(* PLC project marvel_thermoVac, Institute of Astronomy Onto 0.0.1 *)
(* stored: creationDateTime 2025-01-01T00:00:00.0, modificationDateTime 2025-01-01T00:00:00.0 *)

{attribute 'qualified_only'}
TYPE TempControlStates : (idle := 0, warming_up := 1, unstable := 2, controlled := 3);
END_TYPE

{attribute 'qualified_only'}
TYPE TempControlStatus : (unknown := 0, invalid_model := 1, idle := 2, warming_up := 3, unstable := 4, controlled := 5) BYTE;
END_TYPE

TYPE InnerRoomControlParts : STRUCT
  {attribute 'TcHmiSymbol.Show'}
  tpT1 : TempMeasurement;  (* 1st temp sensor *)
  {attribute 'TcHmiSymbol.Show'}
  tpT2 : TempMeasurement;  (* 2nd temp sensor *)
  {attribute 'TcHmiSymbol.Show'}
  tpT3 : TempMeasurement;  (* 3rd temp sensor *)
  {attribute 'TcHmiSymbol.Show'}
  tpT4 : TempMeasurement;  (* 4th temp sensor *)
END_STRUCT;
END_TYPE

TYPE VesselControlParts : STRUCT
  {attribute 'TcHmiSymbol.Show'}
  tpLegNE : TempMeasurement;  (* Leg NE *)
  {attribute 'TcHmiSymbol.Show'}
  tpLegNW : TempMeasurement;  (* Leg NW *)
  {attribute 'TcHmiSymbol.Show'}
  tpLegSE : TempMeasurement;  (* Leg SE *)
  {attribute 'TcHmiSymbol.Show'}
  tpLegSW : TempMeasurement;  (* Leg SW *)
  {attribute 'TcHmiSymbol.Show'}
  tpLegTopNE : TempMeasurement;  (* Leg Top NE *)
  {attribute 'TcHmiSymbol.Show'}
  tpLegTopNW : TempMeasurement;  (* Leg Top NW *)
  {attribute 'TcHmiSymbol.Show'}
  tpLegTopSE : TempMeasurement;  (* Leg Top SE *)
  {attribute 'TcHmiSymbol.Show'}
  tpLegTopSW : TempMeasurement;  (* Leg Top SW *)
  {attribute 'TcHmiSymbol.Show'}
  tpVesBotNE : TempMeasurement;  (* Vessel Bottom NE *)
  {attribute 'TcHmiSymbol.Show'}
  tpVesBotNW : TempMeasurement;  (* Vessel Bottom NW *)
  {attribute 'TcHmiSymbol.Show'}
  tpVesBotSE : TempMeasurement;  (* Vessel Bottom SE *)
  {attribute 'TcHmiSymbol.Show'}
  tpVesBotSW : TempMeasurement;  (* Vessel Bottom SW *)
  {attribute 'TcHmiSymbol.Show'}
  tpCentre : TempMeasurement;  (* Centre *)
  {attribute 'TcHmiSymbol.Show'}
  tpCentreTH10K : TempMeasurement;  (* Centre TH10K *)
  {attribute 'TcHmiSymbol.Show'}
  tpVesSideN : TempMeasurement;  (* Vessel Side N *)
  {attribute 'TcHmiSymbol.Show'}
  tpVesSideS : TempMeasurement;  (* Vessel Side S *)
  {attribute 'TcHmiSymbol.Show'}
  tpVesSideE : TempMeasurement;  (* Vessel Side E *)
  {attribute 'TcHmiSymbol.Show'}
  tpVesSideW : TempMeasurement;  (* Vessel Side W *)
  {attribute 'TcHmiSymbol.Show'}
  tpVesLidN : TempMeasurement;  (* Vessel Lid N *)
  {attribute 'TcHmiSymbol.Show'}
  tpVesLidS : TempMeasurement;  (* Vessel Lid S *)
  {attribute 'TcHmiSymbol.Show'}
  htLegNE : HeaterControl;  (* Heater control for Leg NE *)
  {attribute 'TcHmiSymbol.Show'}
  htLegNW : HeaterControl;  (* Heater control for Leg NW *)
  {attribute 'TcHmiSymbol.Show'}
  htLegSE : HeaterControl;  (* Heater control for Leg SE *)
  {attribute 'TcHmiSymbol.Show'}
  htLegSW : HeaterControl;  (* Heater control for Leg SW *)
  {attribute 'TcHmiSymbol.Show'}
  htLegTopNE : HeaterControl;  (* Heater control for Leg Top NE *)
  {attribute 'TcHmiSymbol.Show'}
  htLegTopNW : HeaterControl;  (* Heater control for Leg Top NW *)
  {attribute 'TcHmiSymbol.Show'}
  htLegTopSE : HeaterControl;  (* Heater control for Leg Top SE *)
  {attribute 'TcHmiSymbol.Show'}
  htLegTopSW : HeaterControl;  (* Heater control for Leg Top SW *)
  {attribute 'TcHmiSymbol.Show'}
  htVesBotNE : HeaterControl;  (* Heater control for Vessel Bottom NE *)
  {attribute 'TcHmiSymbol.Show'}
  htVesBotNW : HeaterControl;  (* Heater control for Vessel Bottom NW *)
  {attribute 'TcHmiSymbol.Show'}
  htVesBotSE : HeaterControl;  (* Heater control for Vessel Bottom SE *)
  {attribute 'TcHmiSymbol.Show'}
  htVesBotSW : HeaterControl;  (* Heater control for Vessel Bottom SW *)
  {attribute 'TcHmiSymbol.Show'}
  htVesSideN : HeaterControl;  (* Heater control for Vessel Side NE *)
  {attribute 'TcHmiSymbol.Show'}
  htVesSideS : HeaterControl;  (* Heater control for Vessel Side NW *)
  {attribute 'TcHmiSymbol.Show'}
  htVesSideE : HeaterControl;  (* Heater control for Vessel Side SE *)
  {attribute 'TcHmiSymbol.Show'}
  htVesSideW : HeaterControl;  (* Heater control for Vessel Side SW *)
  {attribute 'TcHmiSymbol.Show'}
  htVesLidN : HeaterControl;  (* Heater control for Vessel Lid N *)
  {attribute 'TcHmiSymbol.Show'}
  htVesLidS : HeaterControl;  (* Heater control for Vessel Lid S *)
END_STRUCT;
END_TYPE

TYPE CryoControlParts : STRUCT
  {attribute 'TcHmiSymbol.Show'}
  tpCryoRear : TempMeasurement;  (* temp cryo rear / outside *)
  {attribute 'TcHmiSymbol.Show'}
  htCryoRear : HeaterControl;  (* heater cryo rear / outside *)
END_STRUCT;
END_TYPE

TYPE ThermoControlParts : STRUCT
  {attribute 'TcHmiSymbol.Show'}
  vessel : VesselControl;  (* State machine for the vessel temperature control *)
  {attribute 'TcHmiSymbol.Show'}
  innerRoom : InnerRoomControl;  (* State machine for the inner room temperature control *)
  {attribute 'TcHmiSymbol.Show'}
  configManager : ConfigManager;  (* The config manager (to load/save/activate configuration data) *)
END_STRUCT;
END_TYPE

TYPE HeaterControlProcesses : STRUCT
  {attribute 'TcHmiSymbol.Show'}
  initialize : Process;  (* Initialize the heater *)
  {attribute 'TcHmiSymbol.Show'}
  reset : Process;  (* Reset the heater *)
END_STRUCT;
END_TYPE

TYPE OuterRoomControlProcesses : STRUCT
  {attribute 'TcHmiSymbol.Show'}
  initialize : Process;  (* Start initializing *)
  {attribute 'TcHmiSymbol.Show'}
  start : Process;  (* Start warming up *)
  {attribute 'TcHmiSymbol.Show'}
  stop : Process;  (* Stop heating *)
  {attribute 'TcHmiSymbol.Show'}
  reset : Process;  (* Reset complete *)
  {attribute 'TcHmiSymbol.Show'}
  lock : Process;  (* Lock the outer room control (e.g. when the outer room is opened) *)
  {attribute 'TcHmiSymbol.Show'}
  unlock : Process;  (* Unlock the outer room control (e.g. when the outer room is closed) *)
END_STRUCT;
END_TYPE

TYPE InnerRoomControlProcesses : STRUCT
  {attribute 'TcHmiSymbol.Show'}
  initialize : Process;  (* Start initializing *)
  {attribute 'TcHmiSymbol.Show'}
  start : Process;  (* Start warming up *)
  {attribute 'TcHmiSymbol.Show'}
  stop : Process;  (* Stop heating *)
  {attribute 'TcHmiSymbol.Show'}
  reset : Process;  (* Reset complete *)
  {attribute 'TcHmiSymbol.Show'}
  lock : Process;  (* Lock the vessel control (e.g. when the vessel is opened) *)
  {attribute 'TcHmiSymbol.Show'}
  unlock : Process;  (* Unlock the vessel control (e.g. when the vessel is closed) *)
END_STRUCT;
END_TYPE

TYPE VesselControlProcesses : STRUCT
  {attribute 'TcHmiSymbol.Show'}
  initialize : Process;  (* Start initializing *)
  {attribute 'TcHmiSymbol.Show'}
  start : Process;  (* Start warming up *)
  {attribute 'TcHmiSymbol.Show'}
  stop : Process;  (* Stop heating *)
  {attribute 'TcHmiSymbol.Show'}
  reset : Process;  (* Reset complete *)
  {attribute 'TcHmiSymbol.Show'}
  lock : Process;  (* Lock the vessel control (e.g. when the vessel is opened) *)
  {attribute 'TcHmiSymbol.Show'}
  unlock : Process;  (* Unlock the vessel control (e.g. when the vessel is closed) *)
END_STRUCT;
END_TYPE

TYPE ShieldControlProcesses : STRUCT
  {attribute 'TcHmiSymbol.Show'}
  initialize : Process;  (* Start initializing *)
  {attribute 'TcHmiSymbol.Show'}
  start : Process;  (* Start warming up *)
  {attribute 'TcHmiSymbol.Show'}
  stop : Process;  (* Stop heating *)
  {attribute 'TcHmiSymbol.Show'}
  reset : Process;  (* Reset complete *)
  {attribute 'TcHmiSymbol.Show'}
  lock : Process;  (* Lock the shield control (e.g. when the shield is opened) *)
  {attribute 'TcHmiSymbol.Show'}
  unlock : Process;  (* Unlock the shield control (e.g. when the shield is closed) *)
END_STRUCT;
END_TYPE

TYPE BenchControlProcesses : STRUCT
  {attribute 'TcHmiSymbol.Show'}
  initialize : Process;  (* Start initializing *)
  {attribute 'TcHmiSymbol.Show'}
  start : Process;  (* Start warming up *)
  {attribute 'TcHmiSymbol.Show'}
  stop : Process;  (* Stop heating *)
  {attribute 'TcHmiSymbol.Show'}
  reset : Process;  (* Reset complete *)
  {attribute 'TcHmiSymbol.Show'}
  lock : Process;  (* Lock the bench control (e.g. when the bench is opened) *)
  {attribute 'TcHmiSymbol.Show'}
  unlock : Process;  (* Unlock the bench control (e.g. when the bench is closed) *)
END_STRUCT;
END_TYPE

TYPE CryoControlProcesses : STRUCT
  {attribute 'TcHmiSymbol.Show'}
  initialize : Process;  (* Start initializing *)
  {attribute 'TcHmiSymbol.Show'}
  start : Process;  (* Start warming up *)
  {attribute 'TcHmiSymbol.Show'}
  stop : Process;  (* Stop heating *)
  {attribute 'TcHmiSymbol.Show'}
  reset : Process;  (* Reset complete *)
  {attribute 'TcHmiSymbol.Show'}
  lock : Process;  (* Lock the bench control (e.g. when the bench is opened) *)
  {attribute 'TcHmiSymbol.Show'}
  unlock : Process;  (* Unlock the bench control (e.g. when the bench is closed) *)
END_STRUCT;
END_TYPE

TYPE ThermoControlProcesses : STRUCT
  {attribute 'TcHmiSymbol.Show'}
  initialize : Process;  (* Start initializing *)
  {attribute 'TcHmiSymbol.Show'}
  start : Process;  (* Start warming up *)
  {attribute 'TcHmiSymbol.Show'}
  stop : Process;  (* Stop heating *)
  {attribute 'TcHmiSymbol.Show'}
  reset : Process;  (* Reset complete *)
  {attribute 'TcHmiSymbol.Show'}
  lock : Process;  (* Lock the vessel control (e.g. when the vessel is opened) *)
  {attribute 'TcHmiSymbol.Show'}
  unlock : Process;  (* Unlock the vessel control (e.g. when the vessel is closed) *)
END_STRUCT;
END_TYPE

TYPE TempMeasurementStatuses : STRUCT
  {attribute 'OPC.UA.DA' := '1'}
  {attribute 'OPC.UA.DA.Access' := '1'}
  {attribute 'TcHmiSymbol.Show'}
  enabled : EnabledStatus;  (* Is the measurement enabled? *)
  {attribute 'OPC.UA.DA' := '1'}
  {attribute 'OPC.UA.DA.Access' := '1'}
  {attribute 'TcHmiSymbol.Show'}
  health : HealthStatus;  (* Is the measurement OK? *)
  {attribute 'OPC.UA.DA' := '1'}
  {attribute 'OPC.UA.DA.Access' := '1'}
  {attribute 'TcHmiSymbol.Show'}
  alarm : HiHiLoLoAlarmStatus;  (* Alarm status *)
END_STRUCT;
END_TYPE

TYPE HeaterControlStatuses : STRUCT
  {attribute 'OPC.UA.DA' := '1'}
  {attribute 'OPC.UA.DA.Access' := '1'}
  {attribute 'TcHmiSymbol.Show'}
  init : InitializationStatus;
  {attribute 'OPC.UA.DA' := '1'}
  {attribute 'OPC.UA.DA.Access' := '1'}
  {attribute 'TcHmiSymbol.Show'}
  enabled : EnabledStatus;  (* Is the heater enabled? *)
  {attribute 'OPC.UA.DA' := '1'}
  {attribute 'OPC.UA.DA.Access' := '1'}
  {attribute 'TcHmiSymbol.Show'}
  health : HealthStatus;  (* Is the heater healthy? *)
END_STRUCT;
END_TYPE

TYPE OuterRoomControlStatuses : STRUCT
  {attribute 'OPC.UA.DA' := '1'}
  {attribute 'OPC.UA.DA.Access' := '1'}
  {attribute 'TcHmiSymbol.Show'}
  init : InitializationStatus;
  {attribute 'OPC.UA.DA' := '1'}
  {attribute 'OPC.UA.DA.Access' := '1'}
  {attribute 'TcHmiSymbol.Show'}
  health : HealthStatus;  (* Is the outer room healthy? *)
  {attribute 'OPC.UA.DA' := '1'}
  {attribute 'OPC.UA.DA.Access' := '1'}
  {attribute 'TcHmiSymbol.Show'}
  control : TempControlStatus;  (* Actual state of the outer room *)
  {attribute 'OPC.UA.DA' := '1'}
  {attribute 'OPC.UA.DA.Access' := '1'}
  {attribute 'TcHmiSymbol.Show'}
  busy : BusyStatus;  (* Is the outer room busy with a procedure? *)
END_STRUCT;
END_TYPE

TYPE InnerRoomControlStatuses : STRUCT
  {attribute 'OPC.UA.DA' := '1'}
  {attribute 'OPC.UA.DA.Access' := '1'}
  {attribute 'TcHmiSymbol.Show'}
  init : InitializationStatus;
  {attribute 'OPC.UA.DA' := '1'}
  {attribute 'OPC.UA.DA.Access' := '1'}
  {attribute 'TcHmiSymbol.Show'}
  health : HealthStatus;  (* Is the vessel healthy? *)
  {attribute 'OPC.UA.DA' := '1'}
  {attribute 'OPC.UA.DA.Access' := '1'}
  {attribute 'TcHmiSymbol.Show'}
  control : TempControlStatus;  (* Actual state of the vessel *)
  {attribute 'OPC.UA.DA' := '1'}
  {attribute 'OPC.UA.DA.Access' := '1'}
  {attribute 'TcHmiSymbol.Show'}
  busy : BusyStatus;  (* Is the vessel busy with a procedure? *)
END_STRUCT;
END_TYPE

TYPE VesselControlStatuses : STRUCT
  {attribute 'OPC.UA.DA' := '1'}
  {attribute 'OPC.UA.DA.Access' := '1'}
  {attribute 'TcHmiSymbol.Show'}
  init : InitializationStatus;
  {attribute 'OPC.UA.DA' := '1'}
  {attribute 'OPC.UA.DA.Access' := '1'}
  {attribute 'TcHmiSymbol.Show'}
  health : HealthStatus;  (* Is the vessel healthy? *)
  {attribute 'OPC.UA.DA' := '1'}
  {attribute 'OPC.UA.DA.Access' := '1'}
  {attribute 'TcHmiSymbol.Show'}
  control : TempControlStatus;  (* Actual state of the vessel *)
  {attribute 'OPC.UA.DA' := '1'}
  {attribute 'OPC.UA.DA.Access' := '1'}
  {attribute 'TcHmiSymbol.Show'}
  busy : BusyStatus;  (* Is the vessel busy with a procedure? *)
END_STRUCT;
END_TYPE

TYPE ShieldControlStatuses : STRUCT
  {attribute 'OPC.UA.DA' := '1'}
  {attribute 'OPC.UA.DA.Access' := '1'}
  {attribute 'TcHmiSymbol.Show'}
  init : InitializationStatus;
  {attribute 'OPC.UA.DA' := '1'}
  {attribute 'OPC.UA.DA.Access' := '1'}
  {attribute 'TcHmiSymbol.Show'}
  health : HealthStatus;  (* Is the shield healthy? *)
  {attribute 'OPC.UA.DA' := '1'}
  {attribute 'OPC.UA.DA.Access' := '1'}
  {attribute 'TcHmiSymbol.Show'}
  control : TempControlStatus;  (* Actual state of the shield *)
  {attribute 'OPC.UA.DA' := '1'}
  {attribute 'OPC.UA.DA.Access' := '1'}
  {attribute 'TcHmiSymbol.Show'}
  busy : BusyStatus;  (* Is the shield busy with a procedure? *)
END_STRUCT;
END_TYPE

TYPE BenchControlStatuses : STRUCT
  {attribute 'OPC.UA.DA' := '1'}
  {attribute 'OPC.UA.DA.Access' := '1'}
  {attribute 'TcHmiSymbol.Show'}
  init : InitializationStatus;
  {attribute 'OPC.UA.DA' := '1'}
  {attribute 'OPC.UA.DA.Access' := '1'}
  {attribute 'TcHmiSymbol.Show'}
  health : HealthStatus;  (* Is the bench healthy? *)
  {attribute 'OPC.UA.DA' := '1'}
  {attribute 'OPC.UA.DA.Access' := '1'}
  {attribute 'TcHmiSymbol.Show'}
  control : TempControlStatus;  (* Actual state of the bench *)
  {attribute 'OPC.UA.DA' := '1'}
  {attribute 'OPC.UA.DA.Access' := '1'}
  {attribute 'TcHmiSymbol.Show'}
  busy : BusyStatus;  (* Is the bench busy with a procedure? *)
END_STRUCT;
END_TYPE

TYPE CryoControlStatuses : STRUCT
  {attribute 'OPC.UA.DA' := '1'}
  {attribute 'OPC.UA.DA.Access' := '1'}
  {attribute 'TcHmiSymbol.Show'}
  init : InitializationStatus;
  {attribute 'OPC.UA.DA' := '1'}
  {attribute 'OPC.UA.DA.Access' := '1'}
  {attribute 'TcHmiSymbol.Show'}
  health : HealthStatus;  (* Is the bench healthy? *)
  {attribute 'OPC.UA.DA' := '1'}
  {attribute 'OPC.UA.DA.Access' := '1'}
  {attribute 'TcHmiSymbol.Show'}
  control : TempControlStatus;  (* Actual state of the bench *)
  {attribute 'OPC.UA.DA' := '1'}
  {attribute 'OPC.UA.DA.Access' := '1'}
  {attribute 'TcHmiSymbol.Show'}
  busy : BusyStatus;  (* Is the bench busy with a procedure? *)
END_STRUCT;
END_TYPE

TYPE ThermoControlStatuses : STRUCT
  {attribute 'OPC.UA.DA' := '1'}
  {attribute 'OPC.UA.DA.Access' := '1'}
  {attribute 'TcHmiSymbol.Show'}
  init : InitializationStatus;
  {attribute 'OPC.UA.DA' := '1'}
  {attribute 'OPC.UA.DA.Access' := '1'}
  {attribute 'TcHmiSymbol.Show'}
  health : HealthStatus;  (* Is the vessel healthy? *)
  {attribute 'OPC.UA.DA' := '1'}
  {attribute 'OPC.UA.DA.Access' := '1'}
  {attribute 'TcHmiSymbol.Show'}
  control : TempControlStatus;  (* Actual state of the vessel *)
  {attribute 'OPC.UA.DA' := '1'}
  {attribute 'OPC.UA.DA.Access' := '1'}
  {attribute 'TcHmiSymbol.Show'}
  busy : BusyStatus;  (* Is the vessel busy with a procedure? *)
END_STRUCT;
END_TYPE

TYPE HeaterConfig : STRUCT
  {attribute 'TcHmiSymbol.Show'}
  enabled : BOOL := TRUE;  (* True if the heater is enabled *)
  {attribute 'TcHmiSymbol.Show'}
  maxPower : LREAL := 100.0;  (* Maximum power of the heater *)
  {attribute 'TcHmiSymbol.Show'}
  Kp : LREAL;  (* proportional gain *)
  {attribute 'TcHmiSymbol.Show'}
  Tn : LREAL;  (* integral gain (in seconds) *)
  {attribute 'TcHmiSymbol.Show'}
  Tv : LREAL;  (* derivative gain D-T1 (in seconds) *)
  {attribute 'TcHmiSymbol.Show'}
  Td : LREAL;  (* derivative damping time D-T1 (in seconds) *)
END_STRUCT;
END_TYPE

TYPE MeasurementConfig2 : STRUCT
  {attribute 'TcHmiSymbol.Show'}
  enabled : BOOL := TRUE;  (* Is the quantity being measured? (Can be false e.g. if the sensor is deliberately not connected (yet).) *)
  {attribute 'TcHmiSymbol.Show'}
  gain : LREAL := 1.0;  (* Gain to be applied to the measured value (default: 1 = no gain) *)
  {attribute 'TcHmiSymbol.Show'}
  offset : LREAL;  (* Offset to be added to the measured value (default: 0 = no offset) *)
END_STRUCT;
END_TYPE

TYPE SimulationConfig : STRUCT
  {attribute 'TcHmiSymbol.Show'}
  ambient : LREAL;  (* starting temp of sensors *)
  {attribute 'TcHmiSymbol.Show'}
  heating : LREAL;  (* heating gain/factor (0-1) *)
  {attribute 'TcHmiSymbol.Show'}
  cooling : LREAL;  (* cooling factor (0-1) *)
  {attribute 'TcHmiSymbol.Show'}
  noise : LREAL;  (* factor (0-1) multiplied with random number (0-1) to create noise in the simulated temperature *)
END_STRUCT;
END_TYPE

TYPE SharedHeaterConfig : STRUCT
  {attribute 'TcHmiSymbol.Show'}
  hihiDeviation : LREAL;  (* max dev from setpoint *)
  {attribute 'TcHmiSymbol.Show'}
  hiDeviation : LREAL;  (* warning dev from setpoint *)
  {attribute 'TcHmiSymbol.Show'}
  maxPower : LREAL := 100.0;  (* Maximum total power of all heaters in percentage *)
  {attribute 'TcHmiSymbol.Show'}
  simulation : SimulationConfig;
END_STRUCT;
END_TYPE

TYPE OuterRoomSharedConfig : STRUCT
  {attribute 'TcHmiSymbol.Show'}
  sensors : HiHiLoLoAlarmConfig;  (* Alarm config for the temperature sensors in the outer room *)
END_STRUCT;
END_TYPE

TYPE InnerRoomSharedConfig : STRUCT
  {attribute 'TcHmiSymbol.Show'}
  sensors : HiHiLoLoAlarmConfig;  (* Alarm config for the temperature sensors in the inner room *)
END_STRUCT;
END_TYPE

TYPE VesselSharedConfig : STRUCT
  {attribute 'TcHmiSymbol.Show'}
  sensors : HiHiLoLoAlarmConfig;  (* Alarm config for the temperature sensors in the vessel *)
  {attribute 'TcHmiSymbol.Show'}
  heaters : SharedHeaterConfig;  (* Shared config for the heaters in the vessel *)
END_STRUCT;
END_TYPE

TYPE ShieldSharedConfig : STRUCT
  {attribute 'TcHmiSymbol.Show'}
  sensors : HiHiLoLoAlarmConfig;  (* Alarm config for the temperature sensors in the shield *)
END_STRUCT;
END_TYPE

TYPE BenchSharedConfig : STRUCT
  {attribute 'TcHmiSymbol.Show'}
  sensors : HiHiLoLoAlarmConfig;  (* Alarm config for the temperature sensors in the bench *)
END_STRUCT;
END_TYPE

TYPE CryoSharedConfig : STRUCT
  {attribute 'TcHmiSymbol.Show'}
  sensors : HiHiLoLoAlarmConfig;  (* Alarm config for the temperature sensors in the cryo *)
  {attribute 'TcHmiSymbol.Show'}
  heaters : SharedHeaterConfig;  (* Shared config for the heaters in the cryo *)
END_STRUCT;
END_TYPE

TYPE ThermoSharedConfig : STRUCT
  {attribute 'TcHmiSymbol.Show'}
  bool : BOOL;  (* place holder, shared config currently not used *)
END_STRUCT;
END_TYPE

TYPE OuterRoomConfig : STRUCT
  {attribute 'TcHmiSymbol.Show'}
  shared : OuterRoomSharedConfig;  (* Shared config for the outer room *)
END_STRUCT;
END_TYPE

TYPE InnerRoomConfig : STRUCT
  {attribute 'TcHmiSymbol.Show'}
  tpT1 : MeasurementConfig2;  (* Config for temp sensor T1 *)
  {attribute 'TcHmiSymbol.Show'}
  tpT2 : MeasurementConfig2;  (* Config for temp sensor T2 *)
  {attribute 'TcHmiSymbol.Show'}
  tpT3 : MeasurementConfig2;  (* Config for temp sensor T3 *)
  {attribute 'TcHmiSymbol.Show'}
  tpT4 : MeasurementConfig2;  (* Config for temp sensor T4 *)
  {attribute 'TcHmiSymbol.Show'}
  shared : InnerRoomSharedConfig;  (* Shared config for the inner room *)
END_STRUCT;
END_TYPE

TYPE VesselConfig : STRUCT
  {attribute 'TcHmiSymbol.Show'}
  isSimulated : BOOL;  (* True if the vessel temperature control is in simulation mode *)
  {attribute 'TcHmiSymbol.Show'}
  setPointTarget : LREAL;  (* set point temperature in kelvin *)
  {attribute 'TcHmiSymbol.Show'}
  rampVPos : LREAL;  (* velocity of temperature change in K/s while ramping up *)
  {attribute 'TcHmiSymbol.Show'}
  rampVNeg : LREAL;  (* velocity of temperature change in K/s while ramping down *)
  {attribute 'TcHmiSymbol.Show'}
  rampStart : LREAL;  (* temperature in kelvin at which the ramp starts (e.g. to avoid overshoot) *)
  {attribute 'TcHmiSymbol.Show'}
  hihiDeviation : LREAL;  (* max dev from setpoint for the vessel *)
  {attribute 'TcHmiSymbol.Show'}
  hiDeviation : LREAL;  (* warning dev from setpoint for the vessel *)
  {attribute 'TcHmiSymbol.Show'}
  shared : VesselSharedConfig;  (* Shared config for the vessel *)
  {attribute 'TcHmiSymbol.Show'}
  tpLegNE : MeasurementConfig2;  (* Config for Leg NE *)
  {attribute 'TcHmiSymbol.Show'}
  tpLegNW : MeasurementConfig2;  (* Config for Leg NW *)
  {attribute 'TcHmiSymbol.Show'}
  tpLegSE : MeasurementConfig2;  (* Config for Leg SE *)
  {attribute 'TcHmiSymbol.Show'}
  tpLegSW : MeasurementConfig2;  (* Config for Leg SW *)
  {attribute 'TcHmiSymbol.Show'}
  tpLegTopNE : MeasurementConfig2;  (* Config for Leg Top NE *)
  {attribute 'TcHmiSymbol.Show'}
  tpLegTopNW : MeasurementConfig2;  (* Config for Leg Top NW *)
  {attribute 'TcHmiSymbol.Show'}
  tpLegTopSE : MeasurementConfig2;  (* Config for Leg Top SE *)
  {attribute 'TcHmiSymbol.Show'}
  tpLegTopSW : MeasurementConfig2;  (* Config for Leg Top SW *)
  {attribute 'TcHmiSymbol.Show'}
  tpVesBotNE : MeasurementConfig2;  (* Config for Vessel Bottom NE *)
  {attribute 'TcHmiSymbol.Show'}
  tpVesBotNW : MeasurementConfig2;  (* Config for Vessel Bottom NW *)
  {attribute 'TcHmiSymbol.Show'}
  tpVesBotSE : MeasurementConfig2;  (* Config for Vessel Bottom SE *)
  {attribute 'TcHmiSymbol.Show'}
  tpVesBotSW : MeasurementConfig2;  (* Config for Vessel Bottom SW *)
  {attribute 'TcHmiSymbol.Show'}
  tpCentre : MeasurementConfig2;  (* Config for Centre *)
  {attribute 'TcHmiSymbol.Show'}
  tpCentreTH10K : MeasurementConfig2;  (* Config for Centre TH10K *)
  {attribute 'TcHmiSymbol.Show'}
  tpVesSideN : MeasurementConfig2;  (* Config for Vessel Side N *)
  {attribute 'TcHmiSymbol.Show'}
  tpVesSideS : MeasurementConfig2;  (* Config for Vessel Side S *)
  {attribute 'TcHmiSymbol.Show'}
  tpVesSideE : MeasurementConfig2;  (* Config for Vessel Side E *)
  {attribute 'TcHmiSymbol.Show'}
  tpVesSideW : MeasurementConfig2;  (* Config for Vessel Side W *)
  {attribute 'TcHmiSymbol.Show'}
  tpVesLidN : MeasurementConfig2;  (* Config for Vessel Lid N *)
  {attribute 'TcHmiSymbol.Show'}
  tpVesLidS : MeasurementConfig2;  (* Config for Vessel Lid S *)
  {attribute 'TcHmiSymbol.Show'}
  htLegNE : HeaterConfig;  (* Config for heater Leg NE *)
  {attribute 'TcHmiSymbol.Show'}
  htLegNW : HeaterConfig;  (* Config for heater Leg NW *)
  {attribute 'TcHmiSymbol.Show'}
  htLegSE : HeaterConfig;  (* Config for heater Leg SE *)
  {attribute 'TcHmiSymbol.Show'}
  htLegSW : HeaterConfig;  (* Config for heater Leg SW *)
  {attribute 'TcHmiSymbol.Show'}
  htLegTopNE : HeaterConfig;  (* Config for heater Leg Top NE *)
  {attribute 'TcHmiSymbol.Show'}
  htLegTopNW : HeaterConfig;  (* Config for heater Leg Top NW *)
  {attribute 'TcHmiSymbol.Show'}
  htLegTopSE : HeaterConfig;  (* Config for heater Leg Top SE *)
  {attribute 'TcHmiSymbol.Show'}
  htLegTopSW : HeaterConfig;  (* Config for heater Leg Top SW *)
  {attribute 'TcHmiSymbol.Show'}
  htVesBotNE : HeaterConfig;  (* Config for heater Vessel Bottom NE *)
  {attribute 'TcHmiSymbol.Show'}
  htVesBotNW : HeaterConfig;  (* Config for heater Vessel Bottom NW *)
  {attribute 'TcHmiSymbol.Show'}
  htVesBotSE : HeaterConfig;  (* Config for heater Vessel Bottom SE *)
  {attribute 'TcHmiSymbol.Show'}
  htVesBotSW : HeaterConfig;  (* Config for heater Vessel Bottom SW *)
  {attribute 'TcHmiSymbol.Show'}
  htVesSideN : HeaterConfig;  (* Config for heater Vessel Side NE *)
  {attribute 'TcHmiSymbol.Show'}
  htVesSideS : HeaterConfig;  (* Config for heater Vessel Side NW *)
  {attribute 'TcHmiSymbol.Show'}
  htVesSideE : HeaterConfig;  (* Config for heater Vessel Side SE *)
  {attribute 'TcHmiSymbol.Show'}
  htVesSideW : HeaterConfig;  (* Config for heater Vessel Side SW *)
  {attribute 'TcHmiSymbol.Show'}
  htVesLidN : HeaterConfig;  (* Config for heater Vessel Lid N *)
  {attribute 'TcHmiSymbol.Show'}
  htVesLidS : HeaterConfig;  (* Config for heater Vessel Lid S *)
END_STRUCT;
END_TYPE

TYPE ShieldConfig : STRUCT
  {attribute 'TcHmiSymbol.Show'}
  shared : ShieldSharedConfig;  (* Shared config for the shield *)
END_STRUCT;
END_TYPE

TYPE BenchConfig : STRUCT
  {attribute 'TcHmiSymbol.Show'}
  shared : BenchSharedConfig;  (* Shared config for the bench *)
END_STRUCT;
END_TYPE

TYPE CryoConfig : STRUCT
  {attribute 'TcHmiSymbol.Show'}
  shared : CryoSharedConfig;  (* Shared config for the cryo *)
  {attribute 'TcHmiSymbol.Show'}
  tpCryoRear : MeasurementConfig2;  (* config for sensor cryo rear (outside) *)
  {attribute 'TcHmiSymbol.Show'}
  htCryoRear : HeaterConfig;  (* config for heater cryo rear (outside) *)
END_STRUCT;
END_TYPE

TYPE ThermoConfig : STRUCT
  {attribute 'TcHmiSymbol.Show'}
  outerRoom : OuterRoomConfig;  (* Config for the outer room *)
  {attribute 'TcHmiSymbol.Show'}
  innerRoom : InnerRoomConfig;  (* Config for the inner room *)
  {attribute 'TcHmiSymbol.Show'}
  vessel : VesselConfig;  (* Config for the vessel *)
  {attribute 'TcHmiSymbol.Show'}
  shield : ShieldConfig;  (* Config for the shield *)
  {attribute 'TcHmiSymbol.Show'}
  bench : BenchConfig;  (* Config for the bench *)
  {attribute 'TcHmiSymbol.Show'}
  cryo : CryoConfig;  (* Config for the cryo *)
  {attribute 'TcHmiSymbol.Show'}
  shared : ThermoSharedConfig;  (* Shared config for the thermo system *)
END_STRUCT;
END_TYPE

TYPE M_SM_TempMeasurement : STRUCT
  {attribute 'OPC.UA.DA' := '1'}
  {attribute 'OPC.UA.DA.Access' := '1'}
  {attribute 'TcHmiSymbol.Show'}
  isSimulated : BOOL;
  {attribute 'OPC.UA.DA' := '1'}
  {attribute 'OPC.UA.DA.Access' := '1'}
  {attribute 'TcHmiSymbol.Show'}
  simulatedVal : LREAL;
  {attribute 'OPC.UA.DA' := '1'}
  {attribute 'OPC.UA.DA.Access' := '1'}
  {attribute 'TcHmiSymbol.Show'}
  actualStatus : STRING;
  {attribute 'OPC.UA.DA' := '1'}
  {attribute 'OPC.UA.DA.Access' := '1'}
  {attribute 'TcHmiSymbol.Show'}
  actual : LREAL;
  {attribute 'OPC.UA.DA' := '1'}
  {attribute 'OPC.UA.DA.Access' := '1'}
  {attribute 'TcHmiSymbol.Show'}
  average : LREAL;
  {attribute 'OPC.UA.DA' := '1'}
  {attribute 'OPC.UA.DA.Access' := '1'}
  {attribute 'TcHmiSymbol.Show'}
  error : BOOL;
  {attribute 'OPC.UA.DA' := '1'}
  {attribute 'TcHmiSymbol.Show'}
  stat : TempMeasurementStatuses;
END_STRUCT;
END_TYPE

TYPE M_SM_HeaterControl : STRUCT
  {attribute 'OPC.UA.DA' := '1'}
  {attribute 'OPC.UA.DA.Access' := '1'}
  {attribute 'TcHmiSymbol.Show'}
  setPoint : LREAL;
  {attribute 'OPC.UA.DA' := '1'}
  {attribute 'OPC.UA.DA.Access' := '1'}
  {attribute 'TcHmiSymbol.Show'}
  temp : LREAL;
  {attribute 'OPC.UA.DA' := '1'}
  {attribute 'OPC.UA.DA.Access' := '1'}
  {attribute 'TcHmiSymbol.Show'}
  isSimulated : BOOL;
  {attribute 'OPC.UA.DA' := '1'}
  {attribute 'OPC.UA.DA.Access' := '1'}
  {attribute 'TcHmiSymbol.Show'}
  actualStatus : STRING;
  {attribute 'OPC.UA.DA' := '1'}
  {attribute 'OPC.UA.DA.Access' := '1'}
  {attribute 'TcHmiSymbol.Show'}
  power : LREAL;
  {attribute 'OPC.UA.DA' := '1'}
  {attribute 'OPC.UA.DA.Access' := '1'}
  {attribute 'TcHmiSymbol.Show'}
  active : BOOL;
  {attribute 'OPC.UA.DA' := '1'}
  {attribute 'OPC.UA.DA.Access' := '1'}
  {attribute 'TcHmiSymbol.Show'}
  deviation : LREAL;
  {attribute 'OPC.UA.DA' := '1'}
  {attribute 'OPC.UA.DA.Access' := '1'}
  {attribute 'TcHmiSymbol.Show'}
  isControlled : BOOL;
  {attribute 'OPC.UA.DA' := '1'}
  {attribute 'OPC.UA.DA.Access' := '1'}
  {attribute 'TcHmiSymbol.Show'}
  simTemp : LREAL;
  {attribute 'OPC.UA.DA' := '1'}
  {attribute 'TcHmiSymbol.Show'}
  stat : HeaterControlStatuses;
  {attribute 'OPC.UA.DA' := '1'}
  {attribute 'TcHmiSymbol.Show'}
  proc : M_SM_HeaterControlProcesses;
END_STRUCT;
END_TYPE

TYPE M_SM_OuterRoomControl : STRUCT
  {attribute 'OPC.UA.DA' := '1'}
  {attribute 'OPC.UA.DA.Access' := '1'}
  {attribute 'TcHmiSymbol.Show'}
  actualStatus : STRING;
  {attribute 'OPC.UA.DA' := '1'}
  {attribute 'OPC.UA.DA.Access' := '1'}
  {attribute 'TcHmiSymbol.Show'}
  avgTemp : LREAL;
  {attribute 'OPC.UA.DA' := '1'}
  {attribute 'OPC.UA.DA.Access' := '1'}
  {attribute 'TcHmiSymbol.Show'}
  maxDeviation : LREAL;
  {attribute 'OPC.UA.DA' := '1'}
  {attribute 'OPC.UA.DA.Access' := '1'}
  {attribute 'TcHmiSymbol.Show'}
  avgDeviation : LREAL;
  {attribute 'OPC.UA.DA' := '1'}
  {attribute 'OPC.UA.DA.Access' := '1'}
  {attribute 'TcHmiSymbol.Show'}
  totalPower : LREAL;
  {attribute 'OPC.UA.DA' := '1'}
  {attribute 'OPC.UA.DA.Access' := '1'}
  {attribute 'TcHmiSymbol.Show'}
  avgPower : LREAL;
  {attribute 'OPC.UA.DA' := '1'}
  {attribute 'TcHmiSymbol.Show'}
  stat : OuterRoomControlStatuses;
  {attribute 'OPC.UA.DA' := '1'}
  {attribute 'TcHmiSymbol.Show'}
  proc : M_SM_OuterRoomControlProcesses;
END_STRUCT;
END_TYPE

TYPE M_SM_InnerRoomControl : STRUCT
  {attribute 'OPC.UA.DA' := '1'}
  {attribute 'OPC.UA.DA.Access' := '1'}
  {attribute 'TcHmiSymbol.Show'}
  actualStatus : STRING;
  {attribute 'OPC.UA.DA' := '1'}
  {attribute 'OPC.UA.DA.Access' := '1'}
  {attribute 'TcHmiSymbol.Show'}
  avgTemp : LREAL;
  {attribute 'OPC.UA.DA' := '1'}
  {attribute 'OPC.UA.DA.Access' := '1'}
  {attribute 'TcHmiSymbol.Show'}
  maxDeviation : LREAL;
  {attribute 'OPC.UA.DA' := '1'}
  {attribute 'OPC.UA.DA.Access' := '1'}
  {attribute 'TcHmiSymbol.Show'}
  avgDeviation : LREAL;
  {attribute 'OPC.UA.DA' := '1'}
  {attribute 'OPC.UA.DA.Access' := '1'}
  {attribute 'TcHmiSymbol.Show'}
  totalPower : LREAL;
  {attribute 'OPC.UA.DA' := '1'}
  {attribute 'OPC.UA.DA.Access' := '1'}
  {attribute 'TcHmiSymbol.Show'}
  avgPower : LREAL;
  {attribute 'OPC.UA.DA' := '1'}
  {attribute 'TcHmiSymbol.Show'}
  stat : InnerRoomControlStatuses;
  {attribute 'OPC.UA.DA' := '1'}
  {attribute 'TcHmiSymbol.Show'}
  parts : M_SM_InnerRoomControlParts;
  {attribute 'OPC.UA.DA' := '1'}
  {attribute 'TcHmiSymbol.Show'}
  proc : M_SM_InnerRoomControlProcesses;
END_STRUCT;
END_TYPE

TYPE M_SM_VesselControl : STRUCT
  {attribute 'OPC.UA.DA' := '1'}
  {attribute 'OPC.UA.DA.Access' := '1'}
  {attribute 'TcHmiSymbol.Show'}
  tStatBottomOk : BOOL;
  {attribute 'OPC.UA.DA' := '1'}
  {attribute 'OPC.UA.DA.Access' := '1'}
  {attribute 'TcHmiSymbol.Show'}
  tStatCryoRearOk : BOOL;
  {attribute 'OPC.UA.DA' := '1'}
  {attribute 'OPC.UA.DA.Access' := '1'}
  {attribute 'TcHmiSymbol.Show'}
  tStatLidOk : BOOL;
  {attribute 'OPC.UA.DA' := '1'}
  {attribute 'OPC.UA.DA.Access' := '1'}
  {attribute 'TcHmiSymbol.Show'}
  actualStatus : STRING;
  {attribute 'OPC.UA.DA' := '1'}
  {attribute 'OPC.UA.DA.Access' := '1'}
  {attribute 'TcHmiSymbol.Show'}
  avgTemp : LREAL;
  {attribute 'OPC.UA.DA' := '1'}
  {attribute 'OPC.UA.DA.Access' := '1'}
  {attribute 'TcHmiSymbol.Show'}
  maxDeviation : LREAL;
  {attribute 'OPC.UA.DA' := '1'}
  {attribute 'OPC.UA.DA.Access' := '1'}
  {attribute 'TcHmiSymbol.Show'}
  avgDeviation : LREAL;
  {attribute 'OPC.UA.DA' := '1'}
  {attribute 'OPC.UA.DA.Access' := '1'}
  {attribute 'TcHmiSymbol.Show'}
  totalPower : LREAL;
  {attribute 'OPC.UA.DA' := '1'}
  {attribute 'OPC.UA.DA.Access' := '1'}
  {attribute 'TcHmiSymbol.Show'}
  avgPower : LREAL;
  {attribute 'OPC.UA.DA' := '1'}
  {attribute 'OPC.UA.DA.Access' := '1'}
  {attribute 'TcHmiSymbol.Show'}
  tStatBottomPwr : BOOL;
  {attribute 'OPC.UA.DA' := '1'}
  {attribute 'OPC.UA.DA.Access' := '1'}
  {attribute 'TcHmiSymbol.Show'}
  tStatCryoRearPwr : BOOL;
  {attribute 'OPC.UA.DA' := '1'}
  {attribute 'OPC.UA.DA.Access' := '1'}
  {attribute 'TcHmiSymbol.Show'}
  tStatLidPwr : BOOL;
  {attribute 'OPC.UA.DA' := '1'}
  {attribute 'TcHmiSymbol.Show'}
  stat : VesselControlStatuses;
  {attribute 'OPC.UA.DA' := '1'}
  {attribute 'TcHmiSymbol.Show'}
  parts : M_SM_VesselControlParts;
  {attribute 'OPC.UA.DA' := '1'}
  {attribute 'TcHmiSymbol.Show'}
  proc : M_SM_VesselControlProcesses;
END_STRUCT;
END_TYPE

TYPE M_SM_ShieldControl : STRUCT
  {attribute 'OPC.UA.DA' := '1'}
  {attribute 'OPC.UA.DA.Access' := '1'}
  {attribute 'TcHmiSymbol.Show'}
  actualStatus : STRING;
  {attribute 'OPC.UA.DA' := '1'}
  {attribute 'OPC.UA.DA.Access' := '1'}
  {attribute 'TcHmiSymbol.Show'}
  avgTemp : LREAL;
  {attribute 'OPC.UA.DA' := '1'}
  {attribute 'OPC.UA.DA.Access' := '1'}
  {attribute 'TcHmiSymbol.Show'}
  maxDeviation : LREAL;
  {attribute 'OPC.UA.DA' := '1'}
  {attribute 'OPC.UA.DA.Access' := '1'}
  {attribute 'TcHmiSymbol.Show'}
  avgDeviation : LREAL;
  {attribute 'OPC.UA.DA' := '1'}
  {attribute 'OPC.UA.DA.Access' := '1'}
  {attribute 'TcHmiSymbol.Show'}
  totalPower : LREAL;
  {attribute 'OPC.UA.DA' := '1'}
  {attribute 'OPC.UA.DA.Access' := '1'}
  {attribute 'TcHmiSymbol.Show'}
  avgPower : LREAL;
  {attribute 'OPC.UA.DA' := '1'}
  {attribute 'TcHmiSymbol.Show'}
  stat : ShieldControlStatuses;
  {attribute 'OPC.UA.DA' := '1'}
  {attribute 'TcHmiSymbol.Show'}
  proc : M_SM_ShieldControlProcesses;
END_STRUCT;
END_TYPE

TYPE M_SM_BenchControl : STRUCT
  {attribute 'OPC.UA.DA' := '1'}
  {attribute 'OPC.UA.DA.Access' := '1'}
  {attribute 'TcHmiSymbol.Show'}
  actualStatus : STRING;
  {attribute 'OPC.UA.DA' := '1'}
  {attribute 'OPC.UA.DA.Access' := '1'}
  {attribute 'TcHmiSymbol.Show'}
  avgTemp : LREAL;
  {attribute 'OPC.UA.DA' := '1'}
  {attribute 'OPC.UA.DA.Access' := '1'}
  {attribute 'TcHmiSymbol.Show'}
  maxDeviation : LREAL;
  {attribute 'OPC.UA.DA' := '1'}
  {attribute 'OPC.UA.DA.Access' := '1'}
  {attribute 'TcHmiSymbol.Show'}
  avgDeviation : LREAL;
  {attribute 'OPC.UA.DA' := '1'}
  {attribute 'OPC.UA.DA.Access' := '1'}
  {attribute 'TcHmiSymbol.Show'}
  totalPower : LREAL;
  {attribute 'OPC.UA.DA' := '1'}
  {attribute 'OPC.UA.DA.Access' := '1'}
  {attribute 'TcHmiSymbol.Show'}
  avgPower : LREAL;
  {attribute 'OPC.UA.DA' := '1'}
  {attribute 'TcHmiSymbol.Show'}
  stat : BenchControlStatuses;
  {attribute 'OPC.UA.DA' := '1'}
  {attribute 'TcHmiSymbol.Show'}
  proc : M_SM_BenchControlProcesses;
END_STRUCT;
END_TYPE

TYPE M_SM_CryoControl : STRUCT
  {attribute 'OPC.UA.DA' := '1'}
  {attribute 'OPC.UA.DA.Access' := '1'}
  {attribute 'TcHmiSymbol.Show'}
  actualStatus : STRING;
  {attribute 'OPC.UA.DA' := '1'}
  {attribute 'OPC.UA.DA.Access' := '1'}
  {attribute 'TcHmiSymbol.Show'}
  avgTemp : LREAL;
  {attribute 'OPC.UA.DA' := '1'}
  {attribute 'OPC.UA.DA.Access' := '1'}
  {attribute 'TcHmiSymbol.Show'}
  maxDeviation : LREAL;
  {attribute 'OPC.UA.DA' := '1'}
  {attribute 'OPC.UA.DA.Access' := '1'}
  {attribute 'TcHmiSymbol.Show'}
  avgDeviation : LREAL;
  {attribute 'OPC.UA.DA' := '1'}
  {attribute 'OPC.UA.DA.Access' := '1'}
  {attribute 'TcHmiSymbol.Show'}
  totalPower : LREAL;
  {attribute 'OPC.UA.DA' := '1'}
  {attribute 'OPC.UA.DA.Access' := '1'}
  {attribute 'TcHmiSymbol.Show'}
  avgPower : LREAL;
  {attribute 'OPC.UA.DA' := '1'}
  {attribute 'TcHmiSymbol.Show'}
  stat : CryoControlStatuses;
  {attribute 'OPC.UA.DA' := '1'}
  {attribute 'TcHmiSymbol.Show'}
  parts : M_SM_CryoControlParts;
  {attribute 'OPC.UA.DA' := '1'}
  {attribute 'TcHmiSymbol.Show'}
  proc : M_SM_CryoControlProcesses;
END_STRUCT;
END_TYPE

TYPE M_SM_ThermoControl : STRUCT
  {attribute 'OPC.UA.DA' := '1'}
  {attribute 'OPC.UA.DA.Access' := '3'}
  {attribute 'TcHmiSymbol.Show'}
  editableConfig : ThermoConfig;
  {attribute 'OPC.UA.DA' := '1'}
  {attribute 'OPC.UA.DA.Access' := '1'}
  {attribute 'TcHmiSymbol.Show'}
  actualStatus : STRING;
  {attribute 'OPC.UA.DA' := '1'}
  {attribute 'OPC.UA.DA.Access' := '1'}
  {attribute 'TcHmiSymbol.Show'}
  config : ThermoConfig;
  {attribute 'OPC.UA.DA' := '1'}
  {attribute 'OPC.UA.DA.Access' := '1'}
  {attribute 'TcHmiSymbol.Show'}
  setPointRamped : LREAL;
  {attribute 'OPC.UA.DA' := '1'}
  {attribute 'TcHmiSymbol.Show'}
  stat : ThermoControlStatuses;
  {attribute 'OPC.UA.DA' := '1'}
  {attribute 'TcHmiSymbol.Show'}
  parts : M_SM_ThermoControlParts;
  {attribute 'OPC.UA.DA' := '1'}
  {attribute 'TcHmiSymbol.Show'}
  proc : M_SM_ThermoControlProcesses;
END_STRUCT;
END_TYPE

TYPE M_SM_HeaterControlProcesses : STRUCT
  {attribute 'TcHmiSymbol.Show'}
  initialize : M_Process;
  {attribute 'TcHmiSymbol.Show'}
  reset : M_Process;
END_STRUCT;
END_TYPE

TYPE M_SM_OuterRoomControlProcesses : STRUCT
  {attribute 'TcHmiSymbol.Show'}
  initialize : M_Process;
  {attribute 'TcHmiSymbol.Show'}
  start : M_Process;
  {attribute 'TcHmiSymbol.Show'}
  stop : M_Process;
  {attribute 'TcHmiSymbol.Show'}
  reset : M_Process;
  {attribute 'TcHmiSymbol.Show'}
  lock : M_Process;
  {attribute 'TcHmiSymbol.Show'}
  unlock : M_Process;
END_STRUCT;
END_TYPE

TYPE M_SM_InnerRoomControlParts : STRUCT
  {attribute 'TcHmiSymbol.Show'}
  tpT1 : M_TempMeasurement;
  {attribute 'TcHmiSymbol.Show'}
  tpT2 : M_TempMeasurement;
  {attribute 'TcHmiSymbol.Show'}
  tpT3 : M_TempMeasurement;
  {attribute 'TcHmiSymbol.Show'}
  tpT4 : M_TempMeasurement;
END_STRUCT;
END_TYPE

TYPE M_SM_InnerRoomControlProcesses : STRUCT
  {attribute 'TcHmiSymbol.Show'}
  initialize : M_Process;
  {attribute 'TcHmiSymbol.Show'}
  start : M_Process;
  {attribute 'TcHmiSymbol.Show'}
  stop : M_Process;
  {attribute 'TcHmiSymbol.Show'}
  reset : M_Process;
  {attribute 'TcHmiSymbol.Show'}
  lock : M_Process;
  {attribute 'TcHmiSymbol.Show'}
  unlock : M_Process;
END_STRUCT;
END_TYPE

TYPE M_SM_VesselControlParts : STRUCT
  {attribute 'TcHmiSymbol.Show'}
  tpLegNE : M_TempMeasurement;
  {attribute 'TcHmiSymbol.Show'}
  tpLegNW : M_TempMeasurement;
  {attribute 'TcHmiSymbol.Show'}
  tpLegSE : M_TempMeasurement;
  {attribute 'TcHmiSymbol.Show'}
  tpLegSW : M_TempMeasurement;
  {attribute 'TcHmiSymbol.Show'}
  tpLegTopNE : M_TempMeasurement;
  {attribute 'TcHmiSymbol.Show'}
  tpLegTopNW : M_TempMeasurement;
  {attribute 'TcHmiSymbol.Show'}
  tpLegTopSE : M_TempMeasurement;
  {attribute 'TcHmiSymbol.Show'}
  tpLegTopSW : M_TempMeasurement;
  {attribute 'TcHmiSymbol.Show'}
  tpVesBotNE : M_TempMeasurement;
  {attribute 'TcHmiSymbol.Show'}
  tpVesBotNW : M_TempMeasurement;
  {attribute 'TcHmiSymbol.Show'}
  tpVesBotSE : M_TempMeasurement;
  {attribute 'TcHmiSymbol.Show'}
  tpVesBotSW : M_TempMeasurement;
  {attribute 'TcHmiSymbol.Show'}
  tpCentre : M_TempMeasurement;
  {attribute 'TcHmiSymbol.Show'}
  tpCentreTH10K : M_TempMeasurement;
  {attribute 'TcHmiSymbol.Show'}
  tpVesSideN : M_TempMeasurement;
  {attribute 'TcHmiSymbol.Show'}
  tpVesSideS : M_TempMeasurement;
  {attribute 'TcHmiSymbol.Show'}
  tpVesSideE : M_TempMeasurement;
  {attribute 'TcHmiSymbol.Show'}
  tpVesSideW : M_TempMeasurement;
  {attribute 'TcHmiSymbol.Show'}
  tpVesLidN : M_TempMeasurement;
  {attribute 'TcHmiSymbol.Show'}
  tpVesLidS : M_TempMeasurement;
  {attribute 'TcHmiSymbol.Show'}
  htLegNE : M_HeaterControl;
  {attribute 'TcHmiSymbol.Show'}
  htLegNW : M_HeaterControl;
  {attribute 'TcHmiSymbol.Show'}
  htLegSE : M_HeaterControl;
  {attribute 'TcHmiSymbol.Show'}
  htLegSW : M_HeaterControl;
  {attribute 'TcHmiSymbol.Show'}
  htLegTopNE : M_HeaterControl;
  {attribute 'TcHmiSymbol.Show'}
  htLegTopNW : M_HeaterControl;
  {attribute 'TcHmiSymbol.Show'}
  htLegTopSE : M_HeaterControl;
  {attribute 'TcHmiSymbol.Show'}
  htLegTopSW : M_HeaterControl;
  {attribute 'TcHmiSymbol.Show'}
  htVesBotNE : M_HeaterControl;
  {attribute 'TcHmiSymbol.Show'}
  htVesBotNW : M_HeaterControl;
  {attribute 'TcHmiSymbol.Show'}
  htVesBotSE : M_HeaterControl;
  {attribute 'TcHmiSymbol.Show'}
  htVesBotSW : M_HeaterControl;
  {attribute 'TcHmiSymbol.Show'}
  htVesSideN : M_HeaterControl;
  {attribute 'TcHmiSymbol.Show'}
  htVesSideS : M_HeaterControl;
  {attribute 'TcHmiSymbol.Show'}
  htVesSideE : M_HeaterControl;
  {attribute 'TcHmiSymbol.Show'}
  htVesSideW : M_HeaterControl;
  {attribute 'TcHmiSymbol.Show'}
  htVesLidN : M_HeaterControl;
  {attribute 'TcHmiSymbol.Show'}
  htVesLidS : M_HeaterControl;
END_STRUCT;
END_TYPE

TYPE M_SM_VesselControlProcesses : STRUCT
  {attribute 'TcHmiSymbol.Show'}
  initialize : M_Process;
  {attribute 'TcHmiSymbol.Show'}
  start : M_Process;
  {attribute 'TcHmiSymbol.Show'}
  stop : M_Process;
  {attribute 'TcHmiSymbol.Show'}
  reset : M_Process;
  {attribute 'TcHmiSymbol.Show'}
  lock : M_Process;
  {attribute 'TcHmiSymbol.Show'}
  unlock : M_Process;
END_STRUCT;
END_TYPE

TYPE M_SM_ShieldControlProcesses : STRUCT
  {attribute 'TcHmiSymbol.Show'}
  initialize : M_Process;
  {attribute 'TcHmiSymbol.Show'}
  start : M_Process;
  {attribute 'TcHmiSymbol.Show'}
  stop : M_Process;
  {attribute 'TcHmiSymbol.Show'}
  reset : M_Process;
  {attribute 'TcHmiSymbol.Show'}
  lock : M_Process;
  {attribute 'TcHmiSymbol.Show'}
  unlock : M_Process;
END_STRUCT;
END_TYPE

TYPE M_SM_BenchControlProcesses : STRUCT
  {attribute 'TcHmiSymbol.Show'}
  initialize : M_Process;
  {attribute 'TcHmiSymbol.Show'}
  start : M_Process;
  {attribute 'TcHmiSymbol.Show'}
  stop : M_Process;
  {attribute 'TcHmiSymbol.Show'}
  reset : M_Process;
  {attribute 'TcHmiSymbol.Show'}
  lock : M_Process;
  {attribute 'TcHmiSymbol.Show'}
  unlock : M_Process;
END_STRUCT;
END_TYPE

TYPE M_SM_CryoControlParts : STRUCT
  {attribute 'TcHmiSymbol.Show'}
  tpCryoRear : M_TempMeasurement;
  {attribute 'TcHmiSymbol.Show'}
  htCryoRear : M_HeaterControl;
END_STRUCT;
END_TYPE

TYPE M_SM_CryoControlProcesses : STRUCT
  {attribute 'TcHmiSymbol.Show'}
  initialize : M_Process;
  {attribute 'TcHmiSymbol.Show'}
  start : M_Process;
  {attribute 'TcHmiSymbol.Show'}
  stop : M_Process;
  {attribute 'TcHmiSymbol.Show'}
  reset : M_Process;
  {attribute 'TcHmiSymbol.Show'}
  lock : M_Process;
  {attribute 'TcHmiSymbol.Show'}
  unlock : M_Process;
END_STRUCT;
END_TYPE

TYPE M_SM_ThermoControlParts : STRUCT
  {attribute 'TcHmiSymbol.Show'}
  vessel : M_VesselControl;
  {attribute 'TcHmiSymbol.Show'}
  innerRoom : M_InnerRoomControl;
  {attribute 'TcHmiSymbol.Show'}
  configManager : M_ConfigManager;
END_STRUCT;
END_TYPE

TYPE M_SM_ThermoControlProcesses : STRUCT
  {attribute 'TcHmiSymbol.Show'}
  initialize : M_Process;
  {attribute 'TcHmiSymbol.Show'}
  start : M_Process;
  {attribute 'TcHmiSymbol.Show'}
  stop : M_Process;
  {attribute 'TcHmiSymbol.Show'}
  reset : M_Process;
  {attribute 'TcHmiSymbol.Show'}
  lock : M_Process;
  {attribute 'TcHmiSymbol.Show'}
  unlock : M_Process;
END_STRUCT;
END_TYPE

{attribute 'TcRpcEnable' := '1'}
FUNCTION F_TempControlStatus : TempControlStatus
  VAR_INPUT
    superState : BOOL := TRUE;  (* Super state (TRUE if the super state is active, or if there is no super state) *)
    isControlled : BOOL;  (* True if the vessel is in controlled state *)
    isActive : BOOL;  (* True if the vessel is active (not idle) *)
    isWarmingUp : BOOL;  (* True if the vessel is warming up *)
  END_VAR

              IF NOT(superState) THEN
    F_TempControlStatus := TempControlStatus.unknown;
ELSIF NOT(isActive) THEN
    F_TempControlStatus := TempControlStatus.idle;
ELSIF isActive AND isWarmingUp THEN
    F_TempControlStatus := TempControlStatus.warming_up;
ELSIF isActive AND ((NOT(isWarmingUp)) AND (NOT(isControlled))) THEN
    F_TempControlStatus := TempControlStatus.unstable;
ELSIF isActive AND ((NOT(isWarmingUp)) AND isControlled) THEN
    F_TempControlStatus := TempControlStatus.controlled;
ELSE
    F_TempControlStatus := TempControlStatus.invalid_model;
END_IF;

            
END_FUNCTION

FUNCTION_BLOCK SM_TempMeasurement
  VAR_INPUT
    {attribute 'OPC.UA.DA' := '1'}
    {attribute 'OPC.UA.DA.Access' := '1'}
    isSimulated : BOOL;
    {attribute 'OPC.UA.DA' := '1'}
    {attribute 'OPC.UA.DA.Access' := '1'}
    simulatedVal : LREAL;
    {attribute 'OPC.UA.DA' := '0'}
    rawValue AT %I* : REAL;  (* Measured raw value *)
    {attribute 'OPC.UA.DA' := '0'}
    conversionFactor : LREAL;  (* rawValue * conversionFactor = temperature.degrees.value *)
  END_VAR
  VAR_OUTPUT
    {attribute 'OPC.UA.DA' := '1'}
    {attribute 'OPC.UA.DA.Access' := '1'}
    actualStatus : STRING(50);  (* Current status description *)
    {attribute 'OPC.UA.DA' := '1'}
    {attribute 'OPC.UA.DA.Access' := '1'}
    actual : LREAL;  (* Actual value *)
    {attribute 'OPC.UA.DA' := '1'}
    {attribute 'OPC.UA.DA.Access' := '1'}
    average : LREAL;  (* Moving average value *)
    {attribute 'OPC.UA.DA' := '1'}
    {attribute 'OPC.UA.DA.Access' := '1'}
    error : BOOL;  (* true if there is an error *)
    {attribute 'OPC.UA.DA' := '1'}
    stat : TempMeasurementStatuses;  (* Statuses of the state machine *)
  END_VAR
  VAR_IN_OUT
    {attribute 'OPC.UA.DA' := '0'}
    config_ref : MeasurementConfig2;  (* Reference to the config (alarms in degrees celsius) *)
    {attribute 'OPC.UA.DA' := '0'}
    sharedConfig_ref : HiHiLoLoAlarmConfig;  (* Reference to the alarm config for the sensor *)
  END_VAR

            stat.enabled := F_EnabledStatus(
    superState := TRUE,
    isEnabled := config_ref.enabled);
stat.health := F_HealthStatus(
    superState := stat.enabled = EnabledStatus.enabled,
    isGood := NOT((stat.alarm = HiHiLoLoAlarmStatus.hiHi) OR ((stat.alarm = HiHiLoLoAlarmStatus.loLo) OR error)),
    hasWarning := (stat.alarm = HiHiLoLoAlarmStatus.hi) OR (stat.alarm = HiHiLoLoAlarmStatus.lo));

          

METHOD _copyFromModel_SM_TempMeasurement
  VAR_IN_OUT
    {attribute 'OPC.UA.DA' := '0'}
    model : M_SM_TempMeasurement;
  END_VAR
                  
                
END_METHOD

METHOD _copyToModel_SM_TempMeasurement
  VAR_IN_OUT
    {attribute 'OPC.UA.DA' := '0'}
    model : M_SM_TempMeasurement;
  END_VAR
                  model.isSimulated := THIS^.isSimulated;
model.simulatedVal := THIS^.simulatedVal;
model.actualStatus := THIS^.actualStatus;
model.actual := THIS^.actual;
model.average := THIS^.average;
model.error := THIS^.error;
model.stat := THIS^.stat;

                
END_METHOD
END_FUNCTION_BLOCK

FUNCTION_BLOCK SM_HeaterControl
  VAR_INPUT
    {attribute 'OPC.UA.DA' := '1'}
    {attribute 'OPC.UA.DA.Access' := '1'}
    setPoint : LREAL;  (* Current set point of the heater in kelvin *)
    {attribute 'OPC.UA.DA' := '1'}
    {attribute 'OPC.UA.DA.Access' := '1'}
    temp : LREAL;  (* Associated temperature of the heater in kelvin *)
    {attribute 'OPC.UA.DA' := '1'}
    {attribute 'OPC.UA.DA.Access' := '1'}
    isSimulated : BOOL;
  END_VAR
  VAR_OUTPUT
    {attribute 'OPC.UA.DA' := '1'}
    {attribute 'OPC.UA.DA.Access' := '1'}
    actualStatus : STRING(50);  (* Current status description *)
    {attribute 'OPC.UA.DA' := '1'}
    {attribute 'OPC.UA.DA.Access' := '1'}
    power : LREAL;  (* Current power of the heater in percentage *)
    {attribute 'OPC.UA.DA' := '1'}
    {attribute 'OPC.UA.DA.Access' := '1'}
    active : BOOL;  (* True if the heater is active *)
    {attribute 'OPC.UA.DA' := '1'}
    {attribute 'OPC.UA.DA.Access' := '1'}
    deviation : LREAL;  (* Current error between set point and associated temperature *)
    {attribute 'OPC.UA.DA' := '1'}
    {attribute 'OPC.UA.DA.Access' := '1'}
    isControlled : BOOL;  (* True if the heater is in controlled state *)
    {attribute 'OPC.UA.DA' := '1'}
    {attribute 'OPC.UA.DA.Access' := '1'}
    simTemp : LREAL;  (* Simulated temperature for testing the heater control *)
    {attribute 'OPC.UA.DA' := '1'}
    stat : HeaterControlStatuses;  (* Statuses of the state machine *)
    {attribute 'OPC.UA.DA' := '1'}
    proc : HeaterControlProcesses;  (* Processes of the state machine *)
  END_VAR
  VAR_IN_OUT
    {attribute 'OPC.UA.DA' := '0'}
    config_ref : HeaterConfig;  (* Reference to the heater config *)
    {attribute 'OPC.UA.DA' := '0'}
    sharedConfig_ref : SharedHeaterConfig;  (* Reference to the shared heater config *)
  END_VAR

            stat.enabled := F_EnabledStatus(
    superState := TRUE,
    isEnabled := config_ref.enabled);
proc.initialize( isEnabled := NOT((stat.init = InitializationStatus.shutdown) OR ((stat.init = InitializationStatus.initializingFailed) OR (stat.init = InitializationStatus.initialized))) );
proc.reset( isEnabled := TRUE );

          

METHOD _copyFromModel_SM_HeaterControl
  VAR_IN_OUT
    {attribute 'OPC.UA.DA' := '0'}
    model : M_SM_HeaterControl;
  END_VAR
                  THIS^.proc.initialize._copyFromModel_Process( model := model.proc.initialize );
THIS^.proc.reset._copyFromModel_Process( model := model.proc.reset );

                
END_METHOD

METHOD _copyToModel_SM_HeaterControl
  VAR_IN_OUT
    {attribute 'OPC.UA.DA' := '0'}
    model : M_SM_HeaterControl;
  END_VAR
                  model.setPoint := THIS^.setPoint;
model.temp := THIS^.temp;
model.isSimulated := THIS^.isSimulated;
model.actualStatus := THIS^.actualStatus;
model.power := THIS^.power;
model.active := THIS^.active;
model.deviation := THIS^.deviation;
model.isControlled := THIS^.isControlled;
model.simTemp := THIS^.simTemp;
model.stat := THIS^.stat;
THIS^.proc.initialize._copyToModel_Process( model := model.proc.initialize );
THIS^.proc.reset._copyToModel_Process( model := model.proc.reset );

                
END_METHOD
END_FUNCTION_BLOCK

FUNCTION_BLOCK SM_OuterRoomControl
  VAR_OUTPUT
    {attribute 'OPC.UA.DA' := '1'}
    {attribute 'OPC.UA.DA.Access' := '1'}
    actualStatus : STRING(50);  (* Current status description *)
    {attribute 'OPC.UA.DA' := '1'}
    {attribute 'OPC.UA.DA.Access' := '1'}
    avgTemp : LREAL;  (* Average temperature of the outer room in kelvin *)
    {attribute 'OPC.UA.DA' := '1'}
    {attribute 'OPC.UA.DA.Access' := '1'}
    maxDeviation : LREAL;  (* Maximum deviation of the temperature sensors in kelvin *)
    {attribute 'OPC.UA.DA' := '1'}
    {attribute 'OPC.UA.DA.Access' := '1'}
    avgDeviation : LREAL;  (* Average deviation of the temperature sensors in kelvin *)
    {attribute 'OPC.UA.DA' := '1'}
    {attribute 'OPC.UA.DA.Access' := '1'}
    totalPower : LREAL;  (* Total power of all heaters in percentage *)
    {attribute 'OPC.UA.DA' := '1'}
    {attribute 'OPC.UA.DA.Access' := '1'}
    avgPower : LREAL;  (* Average power of the heaters in percentage *)
    {attribute 'OPC.UA.DA' := '1'}
    stat : OuterRoomControlStatuses;  (* Statuses of the state machine *)
    {attribute 'OPC.UA.DA' := '1'}
    proc : OuterRoomControlProcesses;  (* Processes of the state machine *)
  END_VAR
  VAR_IN_OUT
    {attribute 'OPC.UA.DA' := '0'}
    config_ref : OuterRoomConfig;  (* Active configuration of the outer room *)
    {attribute 'OPC.UA.DA' := '0'}
    sharedConfig_ref : ThermoSharedConfig;  (* Shared config for the thermo system *)
    {attribute 'OPC.UA.DA' := '0'}
    activity_ref : ActivityStatus;  (* Shared activity status *)
    {attribute 'OPC.UA.DA' := '0'}
    services_ref : Services;  (* Shared services *)
    {attribute 'OPC.UA.DA' := '0'}
    operator_ref : OperatorStatus;  (* Shared operator status *)
  END_VAR

            proc.initialize( isEnabled := NOT((stat.init = InitializationStatus.shutdown) OR ((stat.init = InitializationStatus.initializingFailed) OR ((stat.init = InitializationStatus.initialized) OR (stat.init = InitializationStatus.locked)))) );
proc.start();
proc.stop();
proc.reset();
proc.lock();
proc.unlock();

          

METHOD _copyFromModel_SM_OuterRoomControl
  VAR_IN_OUT
    {attribute 'OPC.UA.DA' := '0'}
    model : M_SM_OuterRoomControl;
  END_VAR
                  THIS^.proc.initialize._copyFromModel_Process( model := model.proc.initialize );
THIS^.proc.start._copyFromModel_Process( model := model.proc.start );
THIS^.proc.stop._copyFromModel_Process( model := model.proc.stop );
THIS^.proc.reset._copyFromModel_Process( model := model.proc.reset );
THIS^.proc.lock._copyFromModel_Process( model := model.proc.lock );
THIS^.proc.unlock._copyFromModel_Process( model := model.proc.unlock );

                
END_METHOD

METHOD _copyToModel_SM_OuterRoomControl
  VAR_IN_OUT
    {attribute 'OPC.UA.DA' := '0'}
    model : M_SM_OuterRoomControl;
  END_VAR
                  model.actualStatus := THIS^.actualStatus;
model.avgTemp := THIS^.avgTemp;
model.maxDeviation := THIS^.maxDeviation;
model.avgDeviation := THIS^.avgDeviation;
model.totalPower := THIS^.totalPower;
model.avgPower := THIS^.avgPower;
model.stat := THIS^.stat;
THIS^.proc.initialize._copyToModel_Process( model := model.proc.initialize );
THIS^.proc.start._copyToModel_Process( model := model.proc.start );
THIS^.proc.stop._copyToModel_Process( model := model.proc.stop );
THIS^.proc.reset._copyToModel_Process( model := model.proc.reset );
THIS^.proc.lock._copyToModel_Process( model := model.proc.lock );
THIS^.proc.unlock._copyToModel_Process( model := model.proc.unlock );

                
END_METHOD
END_FUNCTION_BLOCK

FUNCTION_BLOCK SM_InnerRoomControl
  VAR_OUTPUT
    {attribute 'OPC.UA.DA' := '1'}
    {attribute 'OPC.UA.DA.Access' := '1'}
    actualStatus : STRING(50);  (* Current status description *)
    {attribute 'OPC.UA.DA' := '1'}
    {attribute 'OPC.UA.DA.Access' := '1'}
    avgTemp : LREAL;  (* Average temperature of the inner room in kelvin *)
    {attribute 'OPC.UA.DA' := '1'}
    {attribute 'OPC.UA.DA.Access' := '1'}
    maxDeviation : LREAL;  (* Maximum deviation of the temperature sensors in kelvin *)
    {attribute 'OPC.UA.DA' := '1'}
    {attribute 'OPC.UA.DA.Access' := '1'}
    avgDeviation : LREAL;  (* Average deviation of the temperature sensors in kelvin *)
    {attribute 'OPC.UA.DA' := '1'}
    {attribute 'OPC.UA.DA.Access' := '1'}
    totalPower : LREAL;  (* Total power of all heaters in percentage *)
    {attribute 'OPC.UA.DA' := '1'}
    {attribute 'OPC.UA.DA.Access' := '1'}
    avgPower : LREAL;  (* Average power of the heaters in percentage *)
    {attribute 'OPC.UA.DA' := '1'}
    stat : InnerRoomControlStatuses;  (* Statuses of the state machine *)
    {attribute 'OPC.UA.DA' := '1'}
    parts : InnerRoomControlParts;  (* Parts of the state machine *)
    {attribute 'OPC.UA.DA' := '1'}
    proc : InnerRoomControlProcesses;  (* Processes of the state machine *)
  END_VAR
  VAR_IN_OUT
    {attribute 'OPC.UA.DA' := '0'}
    config_ref : InnerRoomConfig;  (* Active configuration of the inner room *)
    {attribute 'OPC.UA.DA' := '0'}
    sharedConfig_ref : ThermoSharedConfig;  (* Shared config for the thermo system *)
    {attribute 'OPC.UA.DA' := '0'}
    activity_ref : ActivityStatus;  (* Shared activity status *)
    {attribute 'OPC.UA.DA' := '0'}
    services_ref : Services;  (* Shared services *)
    {attribute 'OPC.UA.DA' := '0'}
    operator_ref : OperatorStatus;  (* Shared operator status *)
  END_VAR

            parts.tpT1(
    config_ref := config_ref.tpT1,
    sharedConfig_ref := config_ref.shared.sensors);
parts.tpT2(
    config_ref := config_ref.tpT2,
    sharedConfig_ref := config_ref.shared.sensors);
parts.tpT3(
    config_ref := config_ref.tpT3,
    sharedConfig_ref := config_ref.shared.sensors);
parts.tpT4(
    config_ref := config_ref.tpT4,
    sharedConfig_ref := config_ref.shared.sensors);
proc.initialize( isEnabled := NOT((stat.init = InitializationStatus.shutdown) OR ((stat.init = InitializationStatus.initializingFailed) OR ((stat.init = InitializationStatus.initialized) OR (stat.init = InitializationStatus.locked)))) );
proc.start();
proc.stop();
proc.reset();
proc.lock();
proc.unlock();

          

METHOD _copyFromModel_SM_InnerRoomControl
  VAR_IN_OUT
    {attribute 'OPC.UA.DA' := '0'}
    model : M_SM_InnerRoomControl;
  END_VAR
                  THIS^.parts.tpT1._copyFromModel_TempMeasurement( model := model.parts.tpT1 );
THIS^.parts.tpT2._copyFromModel_TempMeasurement( model := model.parts.tpT2 );
THIS^.parts.tpT3._copyFromModel_TempMeasurement( model := model.parts.tpT3 );
THIS^.parts.tpT4._copyFromModel_TempMeasurement( model := model.parts.tpT4 );
THIS^.proc.initialize._copyFromModel_Process( model := model.proc.initialize );
THIS^.proc.start._copyFromModel_Process( model := model.proc.start );
THIS^.proc.stop._copyFromModel_Process( model := model.proc.stop );
THIS^.proc.reset._copyFromModel_Process( model := model.proc.reset );
THIS^.proc.lock._copyFromModel_Process( model := model.proc.lock );
THIS^.proc.unlock._copyFromModel_Process( model := model.proc.unlock );

                
END_METHOD

METHOD _copyToModel_SM_InnerRoomControl
  VAR_IN_OUT
    {attribute 'OPC.UA.DA' := '0'}
    model : M_SM_InnerRoomControl;
  END_VAR
                  model.actualStatus := THIS^.actualStatus;
model.avgTemp := THIS^.avgTemp;
model.maxDeviation := THIS^.maxDeviation;
model.avgDeviation := THIS^.avgDeviation;
model.totalPower := THIS^.totalPower;
model.avgPower := THIS^.avgPower;
model.stat := THIS^.stat;
THIS^.parts.tpT1._copyToModel_TempMeasurement( model := model.parts.tpT1 );
THIS^.parts.tpT2._copyToModel_TempMeasurement( model := model.parts.tpT2 );
THIS^.parts.tpT3._copyToModel_TempMeasurement( model := model.parts.tpT3 );
THIS^.parts.tpT4._copyToModel_TempMeasurement( model := model.parts.tpT4 );
THIS^.proc.initialize._copyToModel_Process( model := model.proc.initialize );
THIS^.proc.start._copyToModel_Process( model := model.proc.start );
THIS^.proc.stop._copyToModel_Process( model := model.proc.stop );
THIS^.proc.reset._copyToModel_Process( model := model.proc.reset );
THIS^.proc.lock._copyToModel_Process( model := model.proc.lock );
THIS^.proc.unlock._copyToModel_Process( model := model.proc.unlock );

                
END_METHOD
END_FUNCTION_BLOCK

FUNCTION_BLOCK SM_VesselControl
  VAR_INPUT
    {attribute 'OPC.UA.DA' := '1'}
    {attribute 'OPC.UA.DA.Access' := '1'}
    tStatBottomOk AT %I* : BOOL;  (* State of the thermostat switch at the vessel bottom *)
    {attribute 'OPC.UA.DA' := '1'}
    {attribute 'OPC.UA.DA.Access' := '1'}
    tStatCryoRearOk AT %I* : BOOL;  (* State of the thermostat switch at the cryo rear *)
    {attribute 'OPC.UA.DA' := '1'}
    {attribute 'OPC.UA.DA.Access' := '1'}
    tStatLidOk AT %I* : BOOL;  (* State of the thermostat switch at the lid top *)
  END_VAR
  VAR_OUTPUT
    {attribute 'OPC.UA.DA' := '1'}
    {attribute 'OPC.UA.DA.Access' := '1'}
    actualStatus : STRING(50);  (* Current status description *)
    {attribute 'OPC.UA.DA' := '1'}
    {attribute 'OPC.UA.DA.Access' := '1'}
    avgTemp : LREAL;  (* Average temperature of the vessel in kelvin *)
    {attribute 'OPC.UA.DA' := '1'}
    {attribute 'OPC.UA.DA.Access' := '1'}
    maxDeviation : LREAL;  (* Maximum deviation of the temperature sensors in kelvin *)
    {attribute 'OPC.UA.DA' := '1'}
    {attribute 'OPC.UA.DA.Access' := '1'}
    avgDeviation : LREAL;  (* Average deviation of the temperature sensors in kelvin *)
    {attribute 'OPC.UA.DA' := '1'}
    {attribute 'OPC.UA.DA.Access' := '1'}
    totalPower : LREAL;  (* Total power of all heaters in percentage *)
    {attribute 'OPC.UA.DA' := '1'}
    {attribute 'OPC.UA.DA.Access' := '1'}
    avgPower : LREAL;  (* Average power of the heaters in percentage *)
    {attribute 'OPC.UA.DA' := '1'}
    {attribute 'OPC.UA.DA.Access' := '1'}
    tStatBottomPwr AT %Q* : BOOL;  (* Thermostat switch vessel bottom power *)
    {attribute 'OPC.UA.DA' := '1'}
    {attribute 'OPC.UA.DA.Access' := '1'}
    tStatCryoRearPwr AT %Q* : BOOL;  (* Thermostat switch cryo rear power *)
    {attribute 'OPC.UA.DA' := '1'}
    {attribute 'OPC.UA.DA.Access' := '1'}
    tStatLidPwr AT %Q* : BOOL;  (* Thermostat switch lid top power *)
    {attribute 'OPC.UA.DA' := '1'}
    stat : VesselControlStatuses;  (* Statuses of the state machine *)
    {attribute 'OPC.UA.DA' := '1'}
    parts : VesselControlParts;  (* Parts of the state machine *)
    {attribute 'OPC.UA.DA' := '1'}
    proc : VesselControlProcesses;  (* Processes of the state machine *)
  END_VAR
  VAR_IN_OUT
    {attribute 'OPC.UA.DA' := '0'}
    config_ref : VesselConfig;  (* Active configuration of the vessel *)
    {attribute 'OPC.UA.DA' := '0'}
    sharedConfig_ref : ThermoSharedConfig;  (* Shared config for the thermo system *)
    {attribute 'OPC.UA.DA' := '0'}
    activity_ref : ActivityStatus;  (* Shared activity status *)
    {attribute 'OPC.UA.DA' := '0'}
    services_ref : Services;  (* Shared services *)
    {attribute 'OPC.UA.DA' := '0'}
    operator_ref : OperatorStatus;  (* Shared operator status *)
  END_VAR

            parts.tpLegNE(
    config_ref := config_ref.tpLegNE,
    sharedConfig_ref := config_ref.shared.sensors);
parts.tpLegNW(
    config_ref := config_ref.tpLegNW,
    sharedConfig_ref := config_ref.shared.sensors);
parts.tpLegSE(
    config_ref := config_ref.tpLegSE,
    sharedConfig_ref := config_ref.shared.sensors);
parts.tpLegSW(
    config_ref := config_ref.tpLegSW,
    sharedConfig_ref := config_ref.shared.sensors);
parts.tpLegTopNE(
    config_ref := config_ref.tpLegTopNE,
    sharedConfig_ref := config_ref.shared.sensors);
parts.tpLegTopNW(
    config_ref := config_ref.tpLegTopNW,
    sharedConfig_ref := config_ref.shared.sensors);
parts.tpLegTopSE(
    config_ref := config_ref.tpLegTopSE,
    sharedConfig_ref := config_ref.shared.sensors);
parts.tpLegTopSW(
    config_ref := config_ref.tpLegTopSW,
    sharedConfig_ref := config_ref.shared.sensors);
parts.tpVesBotNE(
    config_ref := config_ref.tpVesBotNE,
    sharedConfig_ref := config_ref.shared.sensors);
parts.tpVesBotNW(
    config_ref := config_ref.tpVesBotNW,
    sharedConfig_ref := config_ref.shared.sensors);
parts.tpVesBotSE(
    config_ref := config_ref.tpVesBotSE,
    sharedConfig_ref := config_ref.shared.sensors);
parts.tpVesBotSW(
    config_ref := config_ref.tpVesBotSW,
    sharedConfig_ref := config_ref.shared.sensors);
parts.tpCentre(
    config_ref := config_ref.tpCentre,
    sharedConfig_ref := config_ref.shared.sensors);
parts.tpCentreTH10K(
    config_ref := config_ref.tpCentreTH10K,
    sharedConfig_ref := config_ref.shared.sensors);
parts.tpVesSideN(
    config_ref := config_ref.tpVesSideN,
    sharedConfig_ref := config_ref.shared.sensors);
parts.tpVesSideS(
    config_ref := config_ref.tpVesSideS,
    sharedConfig_ref := config_ref.shared.sensors);
parts.tpVesSideE(
    config_ref := config_ref.tpVesSideE,
    sharedConfig_ref := config_ref.shared.sensors);
parts.tpVesSideW(
    config_ref := config_ref.tpVesSideW,
    sharedConfig_ref := config_ref.shared.sensors);
parts.tpVesLidN(
    config_ref := config_ref.tpVesLidN,
    sharedConfig_ref := config_ref.shared.sensors);
parts.tpVesLidS(
    config_ref := config_ref.tpVesLidS,
    sharedConfig_ref := config_ref.shared.sensors);
parts.htLegNE(
    config_ref := config_ref.htLegNE,
    sharedConfig_ref := config_ref.shared.heaters);
parts.htLegNW(
    config_ref := config_ref.htLegNW,
    sharedConfig_ref := config_ref.shared.heaters);
parts.htLegSE(
    config_ref := config_ref.htLegSE,
    sharedConfig_ref := config_ref.shared.heaters);
parts.htLegSW(
    config_ref := config_ref.htLegSW,
    sharedConfig_ref := config_ref.shared.heaters);
parts.htLegTopNE(
    config_ref := config_ref.htLegTopNE,
    sharedConfig_ref := config_ref.shared.heaters);
parts.htLegTopNW(
    config_ref := config_ref.htLegTopNW,
    sharedConfig_ref := config_ref.shared.heaters);
parts.htLegTopSE(
    config_ref := config_ref.htLegTopSE,
    sharedConfig_ref := config_ref.shared.heaters);
parts.htLegTopSW(
    config_ref := config_ref.htLegTopSW,
    sharedConfig_ref := config_ref.shared.heaters);
parts.htVesBotNE(
    config_ref := config_ref.htVesBotNE,
    sharedConfig_ref := config_ref.shared.heaters);
parts.htVesBotNW(
    config_ref := config_ref.htVesBotNW,
    sharedConfig_ref := config_ref.shared.heaters);
parts.htVesBotSE(
    config_ref := config_ref.htVesBotSE,
    sharedConfig_ref := config_ref.shared.heaters);
parts.htVesBotSW(
    config_ref := config_ref.htVesBotSW,
    sharedConfig_ref := config_ref.shared.heaters);
parts.htVesSideN(
    config_ref := config_ref.htVesSideN,
    sharedConfig_ref := config_ref.shared.heaters);
parts.htVesSideS(
    config_ref := config_ref.htVesSideS,
    sharedConfig_ref := config_ref.shared.heaters);
parts.htVesSideE(
    config_ref := config_ref.htVesSideE,
    sharedConfig_ref := config_ref.shared.heaters);
parts.htVesSideW(
    config_ref := config_ref.htVesSideW,
    sharedConfig_ref := config_ref.shared.heaters);
parts.htVesLidN(
    config_ref := config_ref.htVesLidN,
    sharedConfig_ref := config_ref.shared.heaters);
parts.htVesLidS(
    config_ref := config_ref.htVesLidS,
    sharedConfig_ref := config_ref.shared.heaters);
proc.initialize( isEnabled := NOT((stat.init = InitializationStatus.shutdown) OR ((stat.init = InitializationStatus.initializingFailed) OR ((stat.init = InitializationStatus.initialized) OR (stat.init = InitializationStatus.locked)))) );
proc.start();
proc.stop();
proc.reset();
proc.lock();
proc.unlock();

          

METHOD _copyFromModel_SM_VesselControl
  VAR_IN_OUT
    {attribute 'OPC.UA.DA' := '0'}
    model : M_SM_VesselControl;
  END_VAR
                  THIS^.parts.tpLegNE._copyFromModel_TempMeasurement( model := model.parts.tpLegNE );
THIS^.parts.tpLegNW._copyFromModel_TempMeasurement( model := model.parts.tpLegNW );
THIS^.parts.tpLegSE._copyFromModel_TempMeasurement( model := model.parts.tpLegSE );
THIS^.parts.tpLegSW._copyFromModel_TempMeasurement( model := model.parts.tpLegSW );
THIS^.parts.tpLegTopNE._copyFromModel_TempMeasurement( model := model.parts.tpLegTopNE );
THIS^.parts.tpLegTopNW._copyFromModel_TempMeasurement( model := model.parts.tpLegTopNW );
THIS^.parts.tpLegTopSE._copyFromModel_TempMeasurement( model := model.parts.tpLegTopSE );
THIS^.parts.tpLegTopSW._copyFromModel_TempMeasurement( model := model.parts.tpLegTopSW );
THIS^.parts.tpVesBotNE._copyFromModel_TempMeasurement( model := model.parts.tpVesBotNE );
THIS^.parts.tpVesBotNW._copyFromModel_TempMeasurement( model := model.parts.tpVesBotNW );
THIS^.parts.tpVesBotSE._copyFromModel_TempMeasurement( model := model.parts.tpVesBotSE );
THIS^.parts.tpVesBotSW._copyFromModel_TempMeasurement( model := model.parts.tpVesBotSW );
THIS^.parts.tpCentre._copyFromModel_TempMeasurement( model := model.parts.tpCentre );
THIS^.parts.tpCentreTH10K._copyFromModel_TempMeasurement( model := model.parts.tpCentreTH10K );
THIS^.parts.tpVesSideN._copyFromModel_TempMeasurement( model := model.parts.tpVesSideN );
THIS^.parts.tpVesSideS._copyFromModel_TempMeasurement( model := model.parts.tpVesSideS );
THIS^.parts.tpVesSideE._copyFromModel_TempMeasurement( model := model.parts.tpVesSideE );
THIS^.parts.tpVesSideW._copyFromModel_TempMeasurement( model := model.parts.tpVesSideW );
THIS^.parts.tpVesLidN._copyFromModel_TempMeasurement( model := model.parts.tpVesLidN );
THIS^.parts.tpVesLidS._copyFromModel_TempMeasurement( model := model.parts.tpVesLidS );
THIS^.parts.htLegNE._copyFromModel_HeaterControl( model := model.parts.htLegNE );
THIS^.parts.htLegNW._copyFromModel_HeaterControl( model := model.parts.htLegNW );
THIS^.parts.htLegSE._copyFromModel_HeaterControl( model := model.parts.htLegSE );
THIS^.parts.htLegSW._copyFromModel_HeaterControl( model := model.parts.htLegSW );
THIS^.parts.htLegTopNE._copyFromModel_HeaterControl( model := model.parts.htLegTopNE );
THIS^.parts.htLegTopNW._copyFromModel_HeaterControl( model := model.parts.htLegTopNW );
THIS^.parts.htLegTopSE._copyFromModel_HeaterControl( model := model.parts.htLegTopSE );
THIS^.parts.htLegTopSW._copyFromModel_HeaterControl( model := model.parts.htLegTopSW );
THIS^.parts.htVesBotNE._copyFromModel_HeaterControl( model := model.parts.htVesBotNE );
THIS^.parts.htVesBotNW._copyFromModel_HeaterControl( model := model.parts.htVesBotNW );
THIS^.parts.htVesBotSE._copyFromModel_HeaterControl( model := model.parts.htVesBotSE );
THIS^.parts.htVesBotSW._copyFromModel_HeaterControl( model := model.parts.htVesBotSW );
THIS^.parts.htVesSideN._copyFromModel_HeaterControl( model := model.parts.htVesSideN );
THIS^.parts.htVesSideS._copyFromModel_HeaterControl( model := model.parts.htVesSideS );
THIS^.parts.htVesSideE._copyFromModel_HeaterControl( model := model.parts.htVesSideE );
THIS^.parts.htVesSideW._copyFromModel_HeaterControl( model := model.parts.htVesSideW );
THIS^.parts.htVesLidN._copyFromModel_HeaterControl( model := model.parts.htVesLidN );
THIS^.parts.htVesLidS._copyFromModel_HeaterControl( model := model.parts.htVesLidS );
THIS^.proc.initialize._copyFromModel_Process( model := model.proc.initialize );
THIS^.proc.start._copyFromModel_Process( model := model.proc.start );
THIS^.proc.stop._copyFromModel_Process( model := model.proc.stop );
THIS^.proc.reset._copyFromModel_Process( model := model.proc.reset );
THIS^.proc.lock._copyFromModel_Process( model := model.proc.lock );
THIS^.proc.unlock._copyFromModel_Process( model := model.proc.unlock );

                
END_METHOD

METHOD _copyToModel_SM_VesselControl
  VAR_IN_OUT
    {attribute 'OPC.UA.DA' := '0'}
    model : M_SM_VesselControl;
  END_VAR
                  model.tStatBottomOk := THIS^.tStatBottomOk;
model.tStatCryoRearOk := THIS^.tStatCryoRearOk;
model.tStatLidOk := THIS^.tStatLidOk;
model.actualStatus := THIS^.actualStatus;
model.avgTemp := THIS^.avgTemp;
model.maxDeviation := THIS^.maxDeviation;
model.avgDeviation := THIS^.avgDeviation;
model.totalPower := THIS^.totalPower;
model.avgPower := THIS^.avgPower;
model.tStatBottomPwr := THIS^.tStatBottomPwr;
model.tStatCryoRearPwr := THIS^.tStatCryoRearPwr;
model.tStatLidPwr := THIS^.tStatLidPwr;
model.stat := THIS^.stat;
THIS^.parts.tpLegNE._copyToModel_TempMeasurement( model := model.parts.tpLegNE );
THIS^.parts.tpLegNW._copyToModel_TempMeasurement( model := model.parts.tpLegNW );
THIS^.parts.tpLegSE._copyToModel_TempMeasurement( model := model.parts.tpLegSE );
THIS^.parts.tpLegSW._copyToModel_TempMeasurement( model := model.parts.tpLegSW );
THIS^.parts.tpLegTopNE._copyToModel_TempMeasurement( model := model.parts.tpLegTopNE );
THIS^.parts.tpLegTopNW._copyToModel_TempMeasurement( model := model.parts.tpLegTopNW );
THIS^.parts.tpLegTopSE._copyToModel_TempMeasurement( model := model.parts.tpLegTopSE );
THIS^.parts.tpLegTopSW._copyToModel_TempMeasurement( model := model.parts.tpLegTopSW );
THIS^.parts.tpVesBotNE._copyToModel_TempMeasurement( model := model.parts.tpVesBotNE );
THIS^.parts.tpVesBotNW._copyToModel_TempMeasurement( model := model.parts.tpVesBotNW );
THIS^.parts.tpVesBotSE._copyToModel_TempMeasurement( model := model.parts.tpVesBotSE );
THIS^.parts.tpVesBotSW._copyToModel_TempMeasurement( model := model.parts.tpVesBotSW );
THIS^.parts.tpCentre._copyToModel_TempMeasurement( model := model.parts.tpCentre );
THIS^.parts.tpCentreTH10K._copyToModel_TempMeasurement( model := model.parts.tpCentreTH10K );
THIS^.parts.tpVesSideN._copyToModel_TempMeasurement( model := model.parts.tpVesSideN );
THIS^.parts.tpVesSideS._copyToModel_TempMeasurement( model := model.parts.tpVesSideS );
THIS^.parts.tpVesSideE._copyToModel_TempMeasurement( model := model.parts.tpVesSideE );
THIS^.parts.tpVesSideW._copyToModel_TempMeasurement( model := model.parts.tpVesSideW );
THIS^.parts.tpVesLidN._copyToModel_TempMeasurement( model := model.parts.tpVesLidN );
THIS^.parts.tpVesLidS._copyToModel_TempMeasurement( model := model.parts.tpVesLidS );
THIS^.parts.htLegNE._copyToModel_HeaterControl( model := model.parts.htLegNE );
THIS^.parts.htLegNW._copyToModel_HeaterControl( model := model.parts.htLegNW );
THIS^.parts.htLegSE._copyToModel_HeaterControl( model := model.parts.htLegSE );
THIS^.parts.htLegSW._copyToModel_HeaterControl( model := model.parts.htLegSW );
THIS^.parts.htLegTopNE._copyToModel_HeaterControl( model := model.parts.htLegTopNE );
THIS^.parts.htLegTopNW._copyToModel_HeaterControl( model := model.parts.htLegTopNW );
THIS^.parts.htLegTopSE._copyToModel_HeaterControl( model := model.parts.htLegTopSE );
THIS^.parts.htLegTopSW._copyToModel_HeaterControl( model := model.parts.htLegTopSW );
THIS^.parts.htVesBotNE._copyToModel_HeaterControl( model := model.parts.htVesBotNE );
THIS^.parts.htVesBotNW._copyToModel_HeaterControl( model := model.parts.htVesBotNW );
THIS^.parts.htVesBotSE._copyToModel_HeaterControl( model := model.parts.htVesBotSE );
THIS^.parts.htVesBotSW._copyToModel_HeaterControl( model := model.parts.htVesBotSW );
THIS^.parts.htVesSideN._copyToModel_HeaterControl( model := model.parts.htVesSideN );
THIS^.parts.htVesSideS._copyToModel_HeaterControl( model := model.parts.htVesSideS );
THIS^.parts.htVesSideE._copyToModel_HeaterControl( model := model.parts.htVesSideE );
THIS^.parts.htVesSideW._copyToModel_HeaterControl( model := model.parts.htVesSideW );
THIS^.parts.htVesLidN._copyToModel_HeaterControl( model := model.parts.htVesLidN );
THIS^.parts.htVesLidS._copyToModel_HeaterControl( model := model.parts.htVesLidS );
THIS^.proc.initialize._copyToModel_Process( model := model.proc.initialize );
THIS^.proc.start._copyToModel_Process( model := model.proc.start );
THIS^.proc.stop._copyToModel_Process( model := model.proc.stop );
THIS^.proc.reset._copyToModel_Process( model := model.proc.reset );
THIS^.proc.lock._copyToModel_Process( model := model.proc.lock );
THIS^.proc.unlock._copyToModel_Process( model := model.proc.unlock );

                
END_METHOD
END_FUNCTION_BLOCK

FUNCTION_BLOCK SM_ShieldControl
  VAR_OUTPUT
    {attribute 'OPC.UA.DA' := '1'}
    {attribute 'OPC.UA.DA.Access' := '1'}
    actualStatus : STRING(50);  (* Current status description *)
    {attribute 'OPC.UA.DA' := '1'}
    {attribute 'OPC.UA.DA.Access' := '1'}
    avgTemp : LREAL;  (* Average temperature of the shield in kelvin *)
    {attribute 'OPC.UA.DA' := '1'}
    {attribute 'OPC.UA.DA.Access' := '1'}
    maxDeviation : LREAL;  (* Maximum deviation of the temperature sensors in kelvin *)
    {attribute 'OPC.UA.DA' := '1'}
    {attribute 'OPC.UA.DA.Access' := '1'}
    avgDeviation : LREAL;  (* Average deviation of the temperature sensors in kelvin *)
    {attribute 'OPC.UA.DA' := '1'}
    {attribute 'OPC.UA.DA.Access' := '1'}
    totalPower : LREAL;  (* Total power of all heaters in percentage *)
    {attribute 'OPC.UA.DA' := '1'}
    {attribute 'OPC.UA.DA.Access' := '1'}
    avgPower : LREAL;  (* Average power of the heaters in percentage *)
    {attribute 'OPC.UA.DA' := '1'}
    stat : ShieldControlStatuses;  (* Statuses of the state machine *)
    {attribute 'OPC.UA.DA' := '1'}
    proc : ShieldControlProcesses;  (* Processes of the state machine *)
  END_VAR
  VAR_IN_OUT
    {attribute 'OPC.UA.DA' := '0'}
    config_ref : ShieldConfig;  (* Active configuration of the shield *)
    {attribute 'OPC.UA.DA' := '0'}
    sharedConfig_ref : ThermoSharedConfig;  (* Shared config for the thermo system *)
    {attribute 'OPC.UA.DA' := '0'}
    activity_ref : ActivityStatus;  (* Shared activity status *)
    {attribute 'OPC.UA.DA' := '0'}
    services_ref : Services;  (* Shared services *)
    {attribute 'OPC.UA.DA' := '0'}
    operator_ref : OperatorStatus;  (* Shared operator status *)
  END_VAR

            proc.initialize( isEnabled := NOT((stat.init = InitializationStatus.shutdown) OR ((stat.init = InitializationStatus.initializingFailed) OR ((stat.init = InitializationStatus.initialized) OR (stat.init = InitializationStatus.locked)))) );
proc.start();
proc.stop();
proc.reset();
proc.lock();
proc.unlock();

          

METHOD _copyFromModel_SM_ShieldControl
  VAR_IN_OUT
    {attribute 'OPC.UA.DA' := '0'}
    model : M_SM_ShieldControl;
  END_VAR
                  THIS^.proc.initialize._copyFromModel_Process( model := model.proc.initialize );
THIS^.proc.start._copyFromModel_Process( model := model.proc.start );
THIS^.proc.stop._copyFromModel_Process( model := model.proc.stop );
THIS^.proc.reset._copyFromModel_Process( model := model.proc.reset );
THIS^.proc.lock._copyFromModel_Process( model := model.proc.lock );
THIS^.proc.unlock._copyFromModel_Process( model := model.proc.unlock );

                
END_METHOD

METHOD _copyToModel_SM_ShieldControl
  VAR_IN_OUT
    {attribute 'OPC.UA.DA' := '0'}
    model : M_SM_ShieldControl;
  END_VAR
                  model.actualStatus := THIS^.actualStatus;
model.avgTemp := THIS^.avgTemp;
model.maxDeviation := THIS^.maxDeviation;
model.avgDeviation := THIS^.avgDeviation;
model.totalPower := THIS^.totalPower;
model.avgPower := THIS^.avgPower;
model.stat := THIS^.stat;
THIS^.proc.initialize._copyToModel_Process( model := model.proc.initialize );
THIS^.proc.start._copyToModel_Process( model := model.proc.start );
THIS^.proc.stop._copyToModel_Process( model := model.proc.stop );
THIS^.proc.reset._copyToModel_Process( model := model.proc.reset );
THIS^.proc.lock._copyToModel_Process( model := model.proc.lock );
THIS^.proc.unlock._copyToModel_Process( model := model.proc.unlock );

                
END_METHOD
END_FUNCTION_BLOCK

FUNCTION_BLOCK SM_BenchControl
  VAR_OUTPUT
    {attribute 'OPC.UA.DA' := '1'}
    {attribute 'OPC.UA.DA.Access' := '1'}
    actualStatus : STRING(50);  (* Current status description *)
    {attribute 'OPC.UA.DA' := '1'}
    {attribute 'OPC.UA.DA.Access' := '1'}
    avgTemp : LREAL;  (* Average temperature of the bench in kelvin *)
    {attribute 'OPC.UA.DA' := '1'}
    {attribute 'OPC.UA.DA.Access' := '1'}
    maxDeviation : LREAL;  (* Maximum deviation of the temperature sensors in kelvin *)
    {attribute 'OPC.UA.DA' := '1'}
    {attribute 'OPC.UA.DA.Access' := '1'}
    avgDeviation : LREAL;  (* Average deviation of the temperature sensors in kelvin *)
    {attribute 'OPC.UA.DA' := '1'}
    {attribute 'OPC.UA.DA.Access' := '1'}
    totalPower : LREAL;  (* Total power of all heaters in percentage *)
    {attribute 'OPC.UA.DA' := '1'}
    {attribute 'OPC.UA.DA.Access' := '1'}
    avgPower : LREAL;  (* Average power of the heaters in percentage *)
    {attribute 'OPC.UA.DA' := '1'}
    stat : BenchControlStatuses;  (* Statuses of the state machine *)
    {attribute 'OPC.UA.DA' := '1'}
    proc : BenchControlProcesses;  (* Processes of the state machine *)
  END_VAR
  VAR_IN_OUT
    {attribute 'OPC.UA.DA' := '0'}
    config_ref : BenchConfig;  (* Active configuration of the bench *)
    {attribute 'OPC.UA.DA' := '0'}
    sharedConfig_ref : ThermoSharedConfig;  (* Shared config for the thermo system *)
    {attribute 'OPC.UA.DA' := '0'}
    activity_ref : ActivityStatus;  (* Shared activity status *)
    {attribute 'OPC.UA.DA' := '0'}
    services_ref : Services;  (* Shared services *)
    {attribute 'OPC.UA.DA' := '0'}
    operator_ref : OperatorStatus;  (* Shared operator status *)
  END_VAR

            proc.initialize( isEnabled := NOT((stat.init = InitializationStatus.shutdown) OR ((stat.init = InitializationStatus.initializingFailed) OR ((stat.init = InitializationStatus.initialized) OR (stat.init = InitializationStatus.locked)))) );
proc.start();
proc.stop();
proc.reset();
proc.lock();
proc.unlock();

          

METHOD _copyFromModel_SM_BenchControl
  VAR_IN_OUT
    {attribute 'OPC.UA.DA' := '0'}
    model : M_SM_BenchControl;
  END_VAR
                  THIS^.proc.initialize._copyFromModel_Process( model := model.proc.initialize );
THIS^.proc.start._copyFromModel_Process( model := model.proc.start );
THIS^.proc.stop._copyFromModel_Process( model := model.proc.stop );
THIS^.proc.reset._copyFromModel_Process( model := model.proc.reset );
THIS^.proc.lock._copyFromModel_Process( model := model.proc.lock );
THIS^.proc.unlock._copyFromModel_Process( model := model.proc.unlock );

                
END_METHOD

METHOD _copyToModel_SM_BenchControl
  VAR_IN_OUT
    {attribute 'OPC.UA.DA' := '0'}
    model : M_SM_BenchControl;
  END_VAR
                  model.actualStatus := THIS^.actualStatus;
model.avgTemp := THIS^.avgTemp;
model.maxDeviation := THIS^.maxDeviation;
model.avgDeviation := THIS^.avgDeviation;
model.totalPower := THIS^.totalPower;
model.avgPower := THIS^.avgPower;
model.stat := THIS^.stat;
THIS^.proc.initialize._copyToModel_Process( model := model.proc.initialize );
THIS^.proc.start._copyToModel_Process( model := model.proc.start );
THIS^.proc.stop._copyToModel_Process( model := model.proc.stop );
THIS^.proc.reset._copyToModel_Process( model := model.proc.reset );
THIS^.proc.lock._copyToModel_Process( model := model.proc.lock );
THIS^.proc.unlock._copyToModel_Process( model := model.proc.unlock );

                
END_METHOD
END_FUNCTION_BLOCK

FUNCTION_BLOCK SM_CryoControl
  VAR_OUTPUT
    {attribute 'OPC.UA.DA' := '1'}
    {attribute 'OPC.UA.DA.Access' := '1'}
    actualStatus : STRING(50);  (* Current status description *)
    {attribute 'OPC.UA.DA' := '1'}
    {attribute 'OPC.UA.DA.Access' := '1'}
    avgTemp : LREAL;  (* Average temperature of the bench in kelvin *)
    {attribute 'OPC.UA.DA' := '1'}
    {attribute 'OPC.UA.DA.Access' := '1'}
    maxDeviation : LREAL;  (* Maximum deviation of the temperature sensors in kelvin *)
    {attribute 'OPC.UA.DA' := '1'}
    {attribute 'OPC.UA.DA.Access' := '1'}
    avgDeviation : LREAL;  (* Average deviation of the temperature sensors in kelvin *)
    {attribute 'OPC.UA.DA' := '1'}
    {attribute 'OPC.UA.DA.Access' := '1'}
    totalPower : LREAL;  (* Total power of all heaters in percentage *)
    {attribute 'OPC.UA.DA' := '1'}
    {attribute 'OPC.UA.DA.Access' := '1'}
    avgPower : LREAL;  (* Average power of the heaters in percentage *)
    {attribute 'OPC.UA.DA' := '1'}
    stat : CryoControlStatuses;  (* Statuses of the state machine *)
    {attribute 'OPC.UA.DA' := '1'}
    parts : CryoControlParts;  (* Parts of the state machine *)
    {attribute 'OPC.UA.DA' := '1'}
    proc : CryoControlProcesses;  (* Processes of the state machine *)
  END_VAR
  VAR_IN_OUT
    {attribute 'OPC.UA.DA' := '0'}
    config_ref : CryoConfig;  (* Active configuration of the bench *)
    {attribute 'OPC.UA.DA' := '0'}
    sharedConfig_ref : ThermoSharedConfig;  (* Shared config for the thermo system *)
    {attribute 'OPC.UA.DA' := '0'}
    activity_ref : ActivityStatus;  (* Shared activity status *)
    {attribute 'OPC.UA.DA' := '0'}
    services_ref : Services;  (* Shared services *)
    {attribute 'OPC.UA.DA' := '0'}
    operator_ref : OperatorStatus;  (* Shared operator status *)
  END_VAR

            parts.tpCryoRear(
    config_ref := config_ref.tpCryoRear,
    sharedConfig_ref := config_ref.shared.sensors);
parts.htCryoRear(
    config_ref := config_ref.htCryoRear,
    sharedConfig_ref := config_ref.shared.heaters);
proc.initialize( isEnabled := NOT((stat.init = InitializationStatus.shutdown) OR ((stat.init = InitializationStatus.initializingFailed) OR ((stat.init = InitializationStatus.initialized) OR (stat.init = InitializationStatus.locked)))) );
proc.start();
proc.stop();
proc.reset();
proc.lock();
proc.unlock();

          

METHOD _copyFromModel_SM_CryoControl
  VAR_IN_OUT
    {attribute 'OPC.UA.DA' := '0'}
    model : M_SM_CryoControl;
  END_VAR
                  THIS^.parts.tpCryoRear._copyFromModel_TempMeasurement( model := model.parts.tpCryoRear );
THIS^.parts.htCryoRear._copyFromModel_HeaterControl( model := model.parts.htCryoRear );
THIS^.proc.initialize._copyFromModel_Process( model := model.proc.initialize );
THIS^.proc.start._copyFromModel_Process( model := model.proc.start );
THIS^.proc.stop._copyFromModel_Process( model := model.proc.stop );
THIS^.proc.reset._copyFromModel_Process( model := model.proc.reset );
THIS^.proc.lock._copyFromModel_Process( model := model.proc.lock );
THIS^.proc.unlock._copyFromModel_Process( model := model.proc.unlock );

                
END_METHOD

METHOD _copyToModel_SM_CryoControl
  VAR_IN_OUT
    {attribute 'OPC.UA.DA' := '0'}
    model : M_SM_CryoControl;
  END_VAR
                  model.actualStatus := THIS^.actualStatus;
model.avgTemp := THIS^.avgTemp;
model.maxDeviation := THIS^.maxDeviation;
model.avgDeviation := THIS^.avgDeviation;
model.totalPower := THIS^.totalPower;
model.avgPower := THIS^.avgPower;
model.stat := THIS^.stat;
THIS^.parts.tpCryoRear._copyToModel_TempMeasurement( model := model.parts.tpCryoRear );
THIS^.parts.htCryoRear._copyToModel_HeaterControl( model := model.parts.htCryoRear );
THIS^.proc.initialize._copyToModel_Process( model := model.proc.initialize );
THIS^.proc.start._copyToModel_Process( model := model.proc.start );
THIS^.proc.stop._copyToModel_Process( model := model.proc.stop );
THIS^.proc.reset._copyToModel_Process( model := model.proc.reset );
THIS^.proc.lock._copyToModel_Process( model := model.proc.lock );
THIS^.proc.unlock._copyToModel_Process( model := model.proc.unlock );

                
END_METHOD
END_FUNCTION_BLOCK

FUNCTION_BLOCK SM_ThermoControl
  VAR_INPUT
    {attribute 'OPC.UA.DA' := '1'}
    {attribute 'OPC.UA.DA.Access' := '3'}
    editableConfig : ThermoConfig;  (* Editable configuration of the thermo system *)
  END_VAR
  VAR_OUTPUT
    {attribute 'OPC.UA.DA' := '1'}
    {attribute 'OPC.UA.DA.Access' := '1'}
    actualStatus : STRING(50);  (* Current status description *)
    {attribute 'OPC.UA.DA' := '1'}
    {attribute 'OPC.UA.DA.Access' := '1'}
    config : ThermoConfig;  (* Active configuration of the thermo system *)
    {attribute 'OPC.UA.DA' := '1'}
    {attribute 'OPC.UA.DA.Access' := '1'}
    setPointRamped : LREAL;  (* Set point temperature in kelvin after ramping *)
    {attribute 'OPC.UA.DA' := '1'}
    stat : ThermoControlStatuses;  (* Statuses of the state machine *)
    {attribute 'OPC.UA.DA' := '1'}
    parts : ThermoControlParts;  (* Parts of the state machine *)
    {attribute 'OPC.UA.DA' := '1'}
    proc : ThermoControlProcesses;  (* Processes of the state machine *)
  END_VAR
  VAR_IN_OUT
    {attribute 'OPC.UA.DA' := '0'}
    activity_ref : ActivityStatus;  (* Shared activity status *)
    {attribute 'OPC.UA.DA' := '0'}
    services_ref : Services;  (* Shared services *)
    {attribute 'OPC.UA.DA' := '0'}
    operator_ref : OperatorStatus;  (* Shared operator status *)
  END_VAR

            parts.vessel(
    activity_ref := activity_ref,
    services_ref := services_ref,
    operator_ref := operator_ref,
    config_ref := config.vessel,
    sharedConfig_ref := config.shared);
parts.innerRoom(
    activity_ref := activity_ref,
    services_ref := services_ref,
    operator_ref := operator_ref,
    config_ref := config.innerRoom,
    sharedConfig_ref := config.shared);
parts.configManager( isEnabled := operator_ref = OperatorStatus.tech );
proc.initialize();
proc.start();
proc.stop();
proc.reset();
proc.lock();
proc.unlock();

          

METHOD _copyFromModel_SM_ThermoControl
  VAR_IN_OUT
    {attribute 'OPC.UA.DA' := '0'}
    model : M_SM_ThermoControl;
  END_VAR
                  THIS^.editableConfig := model.editableConfig;
THIS^.parts.vessel._copyFromModel_VesselControl( model := model.parts.vessel );
THIS^.parts.innerRoom._copyFromModel_InnerRoomControl( model := model.parts.innerRoom );
THIS^.parts.configManager._copyFromModel_ConfigManager( model := model.parts.configManager );
THIS^.proc.initialize._copyFromModel_Process( model := model.proc.initialize );
THIS^.proc.start._copyFromModel_Process( model := model.proc.start );
THIS^.proc.stop._copyFromModel_Process( model := model.proc.stop );
THIS^.proc.reset._copyFromModel_Process( model := model.proc.reset );
THIS^.proc.lock._copyFromModel_Process( model := model.proc.lock );
THIS^.proc.unlock._copyFromModel_Process( model := model.proc.unlock );

                
END_METHOD

METHOD _copyToModel_SM_ThermoControl
  VAR_IN_OUT
    {attribute 'OPC.UA.DA' := '0'}
    model : M_SM_ThermoControl;
  END_VAR
                  model.editableConfig := THIS^.editableConfig;
model.actualStatus := THIS^.actualStatus;
model.config := THIS^.config;
model.setPointRamped := THIS^.setPointRamped;
model.stat := THIS^.stat;
THIS^.parts.vessel._copyToModel_VesselControl( model := model.parts.vessel );
THIS^.parts.innerRoom._copyToModel_InnerRoomControl( model := model.parts.innerRoom );
THIS^.parts.configManager._copyToModel_ConfigManager( model := model.parts.configManager );
THIS^.proc.initialize._copyToModel_Process( model := model.proc.initialize );
THIS^.proc.start._copyToModel_Process( model := model.proc.start );
THIS^.proc.stop._copyToModel_Process( model := model.proc.stop );
THIS^.proc.reset._copyToModel_Process( model := model.proc.reset );
THIS^.proc.lock._copyToModel_Process( model := model.proc.lock );
THIS^.proc.unlock._copyToModel_Process( model := model.proc.unlock );

                
END_METHOD
END_FUNCTION_BLOCK
